(* CODESYS project Codesys_CtrlXCoreDriveConnectUtils
   Author: Riley Duffy
   Company: Open Source
   DefaultNamespace: DriveUtil
   Description: Library to Map Axis Information to it's name
   Title: Axis Info Mapping
   Version: 1.0.0

Project tree, tasks and I/O mapping:
  libraries: CXA_Datalayer, 2.6.20.0 (Bosch Rexroth AG); CXA_Flatbuffers, 0.1.3.2 (Bosch Rexroth AG); CXA_AutomationCore_fbs, 2.6.0.2717 (Bosch Rexroth AG); CXA_MotionCore_fbs, 2.6.0.1 (Bosch Rexroth AG); CXA_MotionSync_fbs, 2.6.0.4874 (Bosch Rexroth AG); CXA_CommonTypes, 1.18.1.0 (Bosch Rexroth AG); Standard, 3.5.18.0 (System); CXA_Utilities, 2.6.2.0 (Bosch Rexroth AG); ADT, 1.0.0 (Open Source); SysExcept, 3.5.17.0 (System)
  function block AxisInfoMap [ST]: Clear, GetAxisInfo, TryGetInfo, TryGetInfoFromAddr, TryPutInfo
  function block AxisInfoMap [ST]
  program AxisMapperPrg [ST]
  program AxisMapperPrg [ST]
  BoschSE_DriveInfoMapping.Sync
  commdata.all
  function block DriveParamBackup [ST]
  function block DriveParamRestore [ST]
  global variables GvlAxisInfo
  global variables GVLAxisInfoMap
  InternHelpers/
    AxisInfo/
      function block AxisInfoContainer [ST]: Get, GetPointer, GetSize, Put
      function block AxisInfoContainer [ST]
      data type typeAxisInfo
    function block AxisInfoMapper [ST]
    function block AxisInfoMapper [ST]
    function block BrowseAxis [ST]
    function block BrowseAxis [ST]
    function block comm_datalayer_DiagMoreInfo [ST]: _assign, _init, addKey, addValue, createDiagMoreInfo, endDiagMoreInfo, getKey, getKeyAsBytePtr, getRootAsDiagMoreInfo, getValue, getValueAsBytePtr, keysCompare, startDiagMoreInfo, verify, verifyDiagMoreInfo
    function block comm_datalayer_Diagnosis [ST]: _assign, _init, addCause, addDetailedDiagnosisCode, addDynamicDescription, addEntity, addMainDiagnosisCode, addMoreInfo, createCauseVector, createDiagnosis, createSortedmoreInfoVector, endDiagnosis, getCause, getCauseLength, getDetailedDiagnosisCode, getDynamicDescription, getDynamicDescriptionAsBytePtr, getEntity, getEntityAsBytePtr, getMainDiagnosisCode, getMoreInfo, getMoreInfoLength, getRootAsDiagnosis, startCauseVector, startDiagnosis, startMoreInfoVector, verify, verifyDiagnosis
    function block comm_datalayer_ProgramTask [ST]: _assign, _init, addId, addProgress, addProgressData, addProgressInfo, addResult, addState, createProgramTask, createSortedprogressDataVector, endProgramTask, getId, getIdAsBytePtr, getProgress, getProgressData, getProgressDataLength, getProgressInfo, getProgressInfoAsBytePtr, getResult, getRootAsProgramTask, getState, keysCompare, startProgramTask, startProgressDataVector, verify, verifyProgramTask
    data type comm_datalayer_ProgramTaskState
    function block comm_datalayer_ProgressData [ST]: _assign, _init, addKey, addValue, createProgressData, endProgressData, getKey, getKeyAsBytePtr, getRootAsProgressData, getValue, getValueAsBytePtr, keysCompare, startProgressData, verify, verifyProgressData
    function block comm_drive_ExportParFile_ExportParFile [ST]: _assign, _init, addBackupType, addFileName, createExportParFile, endExportParFile, getBackupType, getFileName, getFileNameAsBytePtr, getRootAsExportParFile, startExportParFile, verify, verifyExportParFile
    data type comm_drive_ExportParFile_ParametersType
    function block comm_drive_importParameter_ImportParameter [ST]: _assign, _init, addFileName, addSetIndex, createImportParameter, endImportParameter, getFileName, getFileNameAsBytePtr, getRootAsImportParameter, getSetIndex, startImportParameter, verify, verifyImportParameter
    Comparator/
      function block StringCompare [ST]: Compare
      function block StringCompare [ST]
      function block UdintCompare [ST]: Compare
      function block UdintCompare [ST]
    Containers/
      function block DeviceConnectNodeContainer [ST]: Get, GetPointer, GetSize, Put
      function block DeviceConnectNodeContainer [ST]
      function block HashDataContainer [ST]: Get, GetPointer, GetSize, Put
      function block HashDataContainer [ST]
      function block StringDataContainer [ST]: Get, GetPointer, GetSize, Put
      function block StringDataContainer [ST]
      function block UdintContainer [ST]: Get, GetPointer, GetSize, Put
      function block UdintContainer [ST]
    function block DCBrowseForFile [ST]
    data type EN_DRIVE_BACKUP_RESTORE_ERROR
    function block GetAllDriveConnectDevices [ST]
    function block GetAllDriveConnectDevices [ST]
    Hasher/
      function block UdintHash [ST]: Hash
      function block UdintHash [ST]
    function block InitAxisInfoMap [ST]
    function block InitAxisInfoMap [ST]
    function block MapDriveConnect [ST]
    function block MapDriveConnect [ST]
    function StrDecToUDINT [ST]
    function StringHexToUDINT [ST]
    function StringHexToUDINT [ST]
    data type typeDeviceConnectNode
    data type typeDeviceConnectNode
  libDriveUtil.Sync
  function block License_And_Use [ST]
  global variables Param
  global variables Param
  data type typeAxisInfo
*)

// typeAxisInfo
TYPE typeAxisInfo :
STRUCT
	sAxisName: STRING;
	sProfileName: STRING;
	udECatAddr: UDINT;
	sDriveConnectName: STRING;
	iDriveConnectSubDevice: UINT;
END_STRUCT
END_TYPE

// InternHelpers/comm_datalayer_ProgramTaskState
///automatically generated by the FlatBuffers compiler, do not modify
///comm\datalayer
{attribute 'qualified_only' := ''}
TYPE comm_datalayer_ProgramTaskState :
(
	/// task is pending and not been started
	pending := 0,
	/// task finished with failure
	failed := 1,
	/// task is successfully done
	done := 2,
	/// task is running
	running := 3
) BYTE;
END_TYPE

// InternHelpers/comm_drive_ExportParFile_ParametersType
///automatically generated by the FlatBuffers compiler, do not modify
///comm\drive\ExportParFile
{attribute 'qualified_only' := ''}
TYPE comm_drive_ExportParFile_ParametersType :
(
	All := 0,
	Backup := 1,
	Modified := 2
) UDINT;
END_TYPE

// InternHelpers/EN_DRIVE_BACKUP_RESTORE_ERROR
{attribute 'qualified_only' := ''}
{attribute 'strict' := ''}
TYPE EN_DRIVE_BACKUP_RESTORE_ERROR :
(
	OK := 0,
	RequestFailed := 1,
	ProgressReadFailed := 2,
	BackupFailed := 3,
	FileBrowseFailed := 4,
	FileExists := 5,
	DeleteFailed := 6,
	FileNotFound := 7,
	RestoreFailed := 8
);
END_TYPE

// InternHelpers/typeDeviceConnectNode
TYPE typeDeviceConnectNode :
STRUCT
	sNodeName: STRING;
	arSubDevices: ARRAY[0..4] OF STRING;
	uiNumbSubDevices: UINT;
END_STRUCT
END_TYPE

// InternHelpers/typeDeviceConnectNode
{attribute 'hide'}
TYPE typeDeviceConnectNode :
STRUCT
	sNodeName: STRING;
	arSubDevices: ARRAY[0..4] OF STRING;
	uiNumbSubDevices: UINT;
END_STRUCT
END_TYPE

// InternHelpers/AxisInfo/typeAxisInfo
TYPE typeAxisInfo :
STRUCT
	sAxisName: STRING;
	sProfileName: STRING;
	udECatAddr: UDINT;
	sDriveConnectName: STRING;
	iDriveConnectSubDevice: UINT;
END_STRUCT
END_TYPE

// GvlAxisInfo
{attribute 'qualified_only' := ''}
VAR_GLOBAL
	///Map with the Axis Name or EtherCat Address as Key. All Axis used in motion profile auto initialized
	Map: AxisInfoMap;
	///Axis found in the Motion App mapped
	bInitalized: BOOL;
	///Set true to run initialization again, useful if putting non Motion App Drives on map
	bReinitalize: BOOL;
	bClearMap: BOOL;
	///Error Occured during initialization
	Error: BOOL;
	///Only Valid if Error = TRUE
	ErrorID: ERROR_CODE;
	///Only Valid if Error = TRUE
	ErrorIdent: ERROR_STRUCT;
	///Only Valid if Error = TRUE
	ErrorStep: UINT;
END_VAR

// GVLAxisInfoMap
{attribute 'qualified_only'}
(* Interface to the library, Map contains the Drive Axis Info*)
VAR_GLOBAL
	Map : AxisInfoMap; 
	bInitalized :BOOL;
	bReinitalize : BOOL; 
	Error: BOOL;
	ErrorID: ERROR_CODE;
	ErrorIdent: ERROR_STRUCT;
	ErrorStep: UINT;
END_VAR

// Param
{attribute 'parameterlist' := ''}
{attribute 'qualified_only' := ''}
VAR_GLOBAL CONSTANT
	MAX_AXIS: UDINT := 10;
	USE_DRIVE_CONNECT: BOOL := TRUE;
END_VAR

// Param
{attribute 'qualified_only'}
VAR_GLOBAL CONSTANT
	MAX_AXIS : UDINT := 10; 
	USE_DRIVE_CONNECT : BOOL := TRUE; 
END_VAR

// AxisInfoMap
FUNCTION_BLOCK AxisInfoMap
VAR
	Values: AxisInfoContainer;
	Keys: StringDataContainer;
	StrHasher: StringHash;
	StrCompare: StringCompare;
	HashData: HashDataContainer;
	StrHashTable: HashTable := (KeyContainer := Keys, HashDataContainer := HashData, Compareator := StrCompare, Hasher := StrHasher);
	{attribute 'analysis' := '-33'}
	strMap: Map := (KeyContainer := StrHashTable, ValueContainer := Values);
	strValues: StringDataContainer;
	udintKeys: UdintContainer;
	udintHasher: UDintHash;
	udintCompare: UdintCompare;
	HashData2: HashDataContainer;
	UdintHashTable: HashTable := (KeyContainer := udintKeys, HashDataContainer := HashData2, Compareator := udintCompare, Hasher := udintHasher);
	{attribute 'analysis' := '-33'}
	UdintMap: Map := (KeyContainer := UdintHashTable, ValueContainer := strValues);
	stAxisInfo: typeAxisInfo;
END_VAR

METHOD INTERNAL Clear : BOOL
VAR_INPUT
END_VAR
strMap.Clear(); 
UdintMap.Clear();
END_METHOD

METHOD GetAxisInfo : REFERENCE TO typeAxisInfo
VAR_INPUT
	sAxisName: STRING;
END_VAR
strMap.Get(ADR(sAxisName), ADR(stAxisInfo)); 
GetAxisInfo REF= stAxisInfo;
END_METHOD

METHOD TryGetInfo : BOOL
VAR_INPUT
	sAxisName: STRING;
END_VAR
VAR_OUTPUT
	stAxisInfo: typeAxisInfo;
END_VAR
TryGetInfo := strMap.Get(adr(sAxisName),adr(stAxisInfo));
END_METHOD

METHOD TryGetInfoFromAddr : BOOL
VAR_INPUT
	Addr: UDINT;
END_VAR
VAR_OUTPUT
	stAxisInfo: typeAxisInfo;
END_VAR
VAR
	_sAxisName: STRING;
END_VAR
IF UdintMap.Get(ADR(addr),ADR(_sAxisName)) THEN 
	TryGetInfoFromAddr := StrMap.Get(ADR(_sAxisName),ADR(stAxisInfo)); 
ELSE 
	TryGetInfoFromAddr := FALSE; 
END_IF
END_METHOD

METHOD TryPutInfo : BOOL
VAR_INPUT
	sAxisName: STRING;
	stAxisInfo: typeAxisInfo;
END_VAR
TryPutInfo := strMap.Put(ADR(sAxisName),ADR(stAxisInfo)); 
IF stAxisInfo.udECatAddr <> 0 THEN 
	UdintMap.Put(ADR(stAxisInfo.udECatAddr),ADR(sAxisName)); 
END_IF
END_METHOD

END_FUNCTION_BLOCK

// AxisInfoMap
///Axis Info Map used to relate Ethercat Addresses and DeviceConnect Names to axis Name
FUNCTION_BLOCK AxisInfoMap
VAR
	Values: AxisInfoContainer;
	Keys: StringDataContainer;
	StrHasher: StringHash;
	StrCompare: StringCompare;
	HashData: HashDataContainer;
	StrHashTable: HashTable := (KeyContainer := Keys, HashDataContainer := HashData, Compareator := StrCompare, Hasher := StrHasher);
	{attribute 'analysis' := '-33'}
	strMap: Map := (KeyContainer := StrHashTable, ValueContainer := Values);
	strValues: StringDataContainer;
	udintKeys: UdintContainer;
	udintHasher: UDintHash;
	udintCompare: UdintCompare;
	HashData2: HashDataContainer;
	UdintHashTable: HashTable := (KeyContainer := udintKeys, HashDataContainer := HashData2, Compareator := udintCompare, Hasher := udintHasher);
	{attribute 'analysis' := '-33'}
	UdintMap: Map := (KeyContainer := UdintHashTable, ValueContainer := strValues);
	stAxisInfo: typeAxisInfo;
END_VAR

END_FUNCTION_BLOCK

// InternHelpers/AxisInfo/AxisInfoContainer
{attribute 'hide'}
FUNCTION_BLOCK AxisInfoContainer IMPLEMENTS iDataContainer
VAR CONSTANT
	_size : UDINT := TO_UDINT(TO_REAL(Param.MAX_AXIS)* 1.3);
END_VAR 
VAR
	_arBacking: ARRAY[0.._size -1] OF typeAxisInfo;
	_pData: POINTER TO typeAxisInfo;
END_VAR

{attribute 'hide'}
METHOD Get : BOOL
VAR_INPUT
	index: UDINT;
	pData: PVoid;
END_VAR
_pData := pData; 
IF index < _size THEN 
	_pData^ := _arBacking[index]; 
	Get := TRUE;
ELSE 
	Get := FALSE; 
END_IF
END_METHOD

{attribute 'hide'}
METHOD GetPointer : PVoid
VAR_INPUT
	index: UDINT;
END_VAR
IF index < _size THEN 
	GetPointer:= ADR(_arBacking[index]); 
ELSE 
	GetPointer := 0; 
END_IF
END_METHOD

{attribute 'hide'}
METHOD GetSize : UDINT
GetSize := _size;
END_METHOD

{attribute 'hide'}
METHOD Put : BOOL
VAR_INPUT
	index: UDINT;
	pData: PVoid;
END_VAR
_pData := pData; 
IF index < _size THEN 
	_arBacking[index] := _pData^; 
	Put := TRUE; 
ELSE 
	Put := FALSE; 
END_IF
END_METHOD

END_FUNCTION_BLOCK

// InternHelpers/AxisInfo/AxisInfoContainer
FUNCTION_BLOCK AxisInfoContainer IMPLEMENTS iDataContainer
VAR CONSTANT
	_size: UDINT := ANY_TO_UDINT((ANY_TO_REAL(Param.MAX_AXIS) * 1.3));
END_VAR
VAR
	_arBacking: ARRAY[0..(_size - 1)] OF typeAxisInfo;
	_pData: POINTER TO typeAxisInfo;
END_VAR

END_FUNCTION_BLOCK

// InternHelpers/Containers/StringDataContainer
{attribute 'hide'}
{attribute 'no_check' := ''}
FUNCTION_BLOCK StringDataContainer IMPLEMENTS iDataContainer
VAR CONSTANT
	_size : UDINT := TO_UDINT(TO_REAL(Param.MAX_AXIS)* 1.3);
END_VAR 
VAR
	_arBacking: ARRAY[0.._size -1] OF STRING(255);
	_pData: POINTER TO String(255);
END_VAR

{attribute 'hide'}
{attribute 'no_check' := ''}
METHOD Get : BOOL
VAR_INPUT
	index: UDINT;
	pData: PVoid;
END_VAR
_pData := pData; 
IF index < _size THEN 
	_pData^ := _arBacking[index]; 
	Get := TRUE;
ELSE 
	Get := FALSE; 
END_IF
END_METHOD

{attribute 'hide'}
{attribute 'no_check' := ''}
METHOD GetPointer : PVoid
VAR_INPUT
	index: UDINT;
END_VAR
IF index < _size THEN 
	GetPointer:= ADR(_arBacking[index]); 
ELSE 
	GetPointer := 0; 
END_IF
END_METHOD

{attribute 'hide'}
METHOD GetSize : UDINT
GetSize := _size;
END_METHOD

{attribute 'hide'}
{attribute 'no_check' := ''}
METHOD Put : BOOL
VAR_INPUT
	index: UDINT;
	pData: PVoid;
END_VAR
_pData := pData; 
IF index < _size THEN 
	_arBacking[index] := _pData^; 
	Put := TRUE; 
ELSE 
	Put := FALSE; 
END_IF
END_METHOD

END_FUNCTION_BLOCK

// InternHelpers/Containers/StringDataContainer
{attribute 'no_check' := ''}
FUNCTION_BLOCK StringDataContainer IMPLEMENTS iDataContainer
VAR CONSTANT
	_size: UDINT := ANY_TO_UDINT((ANY_TO_REAL(Param.MAX_AXIS) * 1.3));
END_VAR
VAR
	_arBacking: ARRAY[0..(_size - 1)] OF STRING(255);
	_pData: POINTER TO STRING(255);
END_VAR

END_FUNCTION_BLOCK

// InternHelpers/Comparator/StringCompare
{attribute 'hide'}
{attribute 'no_check' := ''}
FUNCTION_BLOCK StringCompare IMPLEMENTS iCompare

{attribute 'hide'}
METHOD Compare : INT
VAR_INPUT
	pData1: PVoid;
	pData2: PVoid;
END_VAR
VAR
	pStr1: POINTER TO STRING := pData1;
	pStr2: POINTER TO STRING := pData2;
END_VAR
IF pStr1^ = pStr2^ THEN 
	Compare := 0; 
ELSE 
	Compare := 1; 
END_IF
END_METHOD

END_FUNCTION_BLOCK

// InternHelpers/Comparator/StringCompare
{attribute 'no_check' := ''}
FUNCTION_BLOCK StringCompare IMPLEMENTS iCompare

END_FUNCTION_BLOCK

// InternHelpers/Containers/HashDataContainer
{attribute 'no_check' := ''}
FUNCTION_BLOCK HashDataContainer IMPLEMENTS iDataContainer
VAR CONSTANT
	_size: UDINT := ANY_TO_UDINT((ANY_TO_REAL(Param.MAX_AXIS) * 1.3));
END_VAR
VAR
	_arBacking: ARRAY[0..(_size - 1)] OF HashData;
	_pData: POINTER TO HashData;
END_VAR

{attribute 'no_check' := ''}
METHOD Get : BOOL
VAR_INPUT
	index: UDINT;
	pData: PVoid;
END_VAR
_pData := pData; 
IF index < _size THEN 
	_pData^ := _arBacking[index]; 
	Get := TRUE;
ELSE 
	Get := FALSE; 
END_IF
END_METHOD

{attribute 'no_check' := ''}
METHOD GetPointer : PVoid
VAR_INPUT
	index: UDINT;
END_VAR
IF index < _size THEN 
	GetPointer:= ADR(_arBacking[index]); 
ELSE 
	GetPointer := 0; 
END_IF
END_METHOD

METHOD GetSize : UDINT
GetSize := _size;
END_METHOD

{attribute 'no_check' := ''}
METHOD Put : BOOL
VAR_INPUT
	index: UDINT;
	pData: PVoid;
END_VAR
_pData := pData; 
IF index < _size THEN 
	_arBacking[index] := _pData^; 
	Put := TRUE; 
ELSE 
	Put := FALSE; 
END_IF
END_METHOD

END_FUNCTION_BLOCK

// InternHelpers/Containers/HashDataContainer
{attribute 'hide'}
{attribute 'no_check' := ''}
FUNCTION_BLOCK HashDataContainer IMPLEMENTS iDataContainer
VAR CONSTANT
	_size : UDINT := TO_UDINT(TO_REAL(Param.MAX_AXIS)* 1.3);
END_VAR 
VAR
	_arBacking: ARRAY[0.._size -1] OF HashData;
	_pData: POINTER TO HashData;
END_VAR

END_FUNCTION_BLOCK

// InternHelpers/Containers/UdintContainer
{attribute 'hide'}
{attribute 'no_check' := ''}
FUNCTION_BLOCK UdintContainer IMPLEMENTS iDataContainer
VAR CONSTANT
	_size : UDINT := TO_UDINT(TO_REAL(Param.MAX_AXIS)* 1.3);
END_VAR 
VAR
	_arBacking: ARRAY[0.._size -1] OF UDINT;
	_pData: POINTER TO UDINT;
END_VAR

{attribute 'hide'}
{attribute 'no_check' := ''}
METHOD Get : BOOL
VAR_INPUT
	index: UDINT;
	pData: PVoid;
END_VAR
_pData := pData; 
IF index < _size THEN 
	_pData^ := _arBacking[index]; 
	Get := TRUE;
ELSE 
	Get := FALSE; 
END_IF
END_METHOD

{attribute 'hide'}
{attribute 'no_check' := ''}
METHOD GetPointer : PVoid
VAR_INPUT
	index: UDINT;
END_VAR
IF index < _size THEN 
	GetPointer:= ADR(_arBacking[index]); 
ELSE 
	GetPointer := 0; 
END_IF
END_METHOD

{attribute 'hide'}
METHOD GetSize : UDINT
GetSize := _size;
END_METHOD

{attribute 'hide'}
{attribute 'no_check' := ''}
METHOD Put : BOOL
VAR_INPUT
	index: UDINT;
	pData: PVoid;
END_VAR
_pData := pData; 
IF index < _size THEN 
	_arBacking[index] := _pData^; 
	Put := TRUE; 
ELSE 
	Put := FALSE; 
END_IF
END_METHOD

END_FUNCTION_BLOCK

// InternHelpers/Containers/UdintContainer
{attribute 'no_check' := ''}
FUNCTION_BLOCK UdintContainer IMPLEMENTS iDataContainer
VAR CONSTANT
	_size: UDINT := ANY_TO_UDINT((ANY_TO_REAL(Param.MAX_AXIS) * 1.3));
END_VAR
VAR
	_arBacking: ARRAY[0..(_size - 1)] OF UDINT;
	_pData: POINTER TO UDINT;
END_VAR

END_FUNCTION_BLOCK

// InternHelpers/Hasher/UdintHash
{attribute 'hide'}
{attribute 'no_check' := ''}
FUNCTION_BLOCK UdintHash IMPLEMENTS iHash

{attribute 'hide'}
METHOD Hash : LINT
VAR_INPUT
	pData: pVoid;
END_VAR
VAR
	ptrUdint: POINTER TO UDINT := pData;
END_VAR
Hash := TO_LINT(ptrUdint^);
END_METHOD

END_FUNCTION_BLOCK

// InternHelpers/Hasher/UdintHash
{attribute 'no_check' := ''}
FUNCTION_BLOCK UdintHash IMPLEMENTS iHash

END_FUNCTION_BLOCK

// InternHelpers/Comparator/UdintCompare
{attribute 'hide'}
{attribute 'no_check' := ''}
FUNCTION_BLOCK UdintCompare IMPLEMENTS iCompare

{attribute 'hide'}
METHOD Compare : INT
VAR_INPUT
	pData1: PVoid;
	pData2: PVoid;
END_VAR
VAR
	pUdint1: POINTER TO UDINT := pData1;
	pUdint2: POINTER TO UDINT := pData2;
END_VAR
IF pUdint1^ = pUdint2^ THEN 
	Compare := 0; 
ELSIF pUdint1^ > pUdint2^ THEN 
	Compare := 1; 
ELSE
	Compare := -1; 
END_IF
END_METHOD

END_FUNCTION_BLOCK

// InternHelpers/Comparator/UdintCompare
{attribute 'no_check' := ''}
FUNCTION_BLOCK UdintCompare IMPLEMENTS iCompare

END_FUNCTION_BLOCK

// AxisMapperPrg
PROGRAM AxisMapperPrg
VAR
	_instAxisMapper: AxisInfoMapper;
	_dlBrowse: CXA_DATALAYER.DL_BrowseNode;
	_sBrowseDevices: STRING(255) := 'devices/drives';
	_bReady: BOOL;
	_fbBootDelay : TON; 
	_bFirstScan : BOOL := TRUE; 
END_VAR

_fbBootDelay(IN := NOT _bFirstScan, PT := T#10s); 
_bFirstScan := FALSE; 
IF NOT _fbBootDelay.Q THEN 
	RETURN
END_IF
IF PARAM.USE_DRIVE_CONNECT AND NOT _bReady THEN 
	_dlBrowse(execute := NOT _bReady, 
			  NodeName := _sBrowseDevices); 
	IF _dlBrowse.Done AND _dlBrowse.ChildPtr = 0 THEN 
		_dlBrowse(execute := FALSE);
	ELSIF _dlBrowse.Done THEN 
		_bReady := TRUE; 
	END_IF
END_IF
IF NOT _bReady THEN 
	RETURN; 
END_IF
_instAxisMapper(bExecute := GvlAxisInfo.bReinitalize OR (NOT GvlAxisInfo.bInitalized AND NOT GvlAxisInfo.Error),
				bUseDriveConnect := Param.USE_DRIVE_CONNECT, 
				instAxisInfoMap := GvlAxisInfo.Map); 
IF _instAxisMapper.bDone THEN 
	GvlAxisInfo.bInitalized := TRUE; 
END_IF
IF GvlAxisInfo.bReinitalize THEN 
	GvlAxisInfo.Error := FALSE; 
END_IF
IF _instAxisMapper.bActive THEN 
	GvlAxisInfo.bInitalized := FALSE; 
END_IF
IF GVLAxisInfo.bClearMap THEN 
	GVLAxisInfo.Map.Clear();
	GvlAxisInfo.bInitalized := FALSE; 
END_IF
IF _instAxisMapper.bError THEN 
	GvlAxisInfo.Error := TRUE; 
END_IF 
IF _instAxisMapper.bError THEN 
	GvlAxisInfo.ErrorID := _instAxisMapper.ErrorID; 
	GvlAxisInfo.ErrorIdent := _instAxisMapper.ErrorIdent; 
	GvlAxisInfo.ErrorStep := _instAxisMapper.ErrorStep; 
END_IF

END_PROGRAM

// AxisMapperPrg
(* Program that searches the configured axis in CtrxCore and gets 
   their Ethercat addresses and Drive Connect info (serial number, drive index)*)
PROGRAM AxisMapperPrg
VAR
	_instAxisMapper : AxisInfoMapper; 
END_VAR
VAR_OUTPUT
	
END_VAR

_instAxisMapper(bExecute := GvlAxisInfoMap.bReinitalize OR NOT GvlAxisInfoMap.bInitalized,
				bUseDriveConnect := Param.USE_DRIVE_CONNECT, 
				instAxisInfoMap := GvlAxisInfoMap.Map); 
IF _instAxisMapper.bDone THEN 
	GvlAxisInfoMap.bInitalized := TRUE; 
END_IF
IF _instAxisMapper.bActive THEN 
	GvlAxisInfoMap.bInitalized := FALSE; 
END_IF

GVLAxisInfoMap.Error := _instAxisMapper.bError; 
IF _instAxisMapper.bError THEN 
	GVLAxisInfoMap.ErrorID := _instAxisMapper.ErrorID; 
	GVLAxisInfoMap.ErrorIdent := _instAxisMapper.ErrorIdent; 
	GVLAxisInfoMap.ErrorStep := _instAxisMapper.ErrorStep; 
END_IF

END_PROGRAM

// InternHelpers/AxisInfoMapper
FUNCTION_BLOCK AxisInfoMapper
VAR_INPUT
	bExecute: BOOL;
	bUseDriveConnect: BOOL;
END_VAR
VAR_IN_OUT
	instAxisInfoMap: AxisInfoMap;
END_VAR
VAR_OUTPUT
	bDone: BOOL;
	bActive: BOOL;
	bError: BOOL;
	ErrorID: ERROR_CODE;
	ErrorIdent: ERROR_STRUCT;
	ErrorStep: UINT;
END_VAR
VAR
	_uiNextState: UINT;
	_uiState: UINT;
	_instInitAxisInfo: InitAxisInfoMap;
	_instMapDriveConnect: MapDriveConnect;
END_VAR
VAR CONSTANT
	IDLE: UINT := 0;
	INIT_AXIS_INFO_MAP: UINT := 1;
	MAP_DRIVE_CONNECT: UINT := 2;
	DONE: UINT := 3;
	ERROR: UINT := 4;
END_VAR

_uiNextState := _uiState; 
CASE _uiState OF 
	IDLE : 
		IF bExecute THEN 
			_uiNextState := INIT_AXIS_INFO_MAP;  
		END_IF
	INIT_AXIS_INFO_MAP: 
		IF _instInitAxisInfo.bError THEN 
			bError := TRUE; 
			ERRORID := _instInitAxisInfo.enErrorID; 
			ErrorIdent := _instInitAxisInfo.enErrorIdent; 
			ErrorStep := INIT_AXIS_INFO_MAP; 
			_uiNextState := ERROR; 
		ELSIF _instInitAxisInfo.bDone THEN 
			IF bUseDriveConnect THEN 
				_uiNextState := MAP_DRIVE_CONNECT; 
			ELSE 
				_uiNextState := DONE; 
			END_IF
		END_IF
	MAP_DRIVE_CONNECT: 
		IF _instMapDriveConnect.bError THEN 
			bError := TRUE; 
			ERRORID := _instMapDriveConnect.enErrorID; 
			ErrorIdent := _instMapDriveConnect.stErrorIdent; 
			ErrorStep := INIT_AXIS_INFO_MAP; 
			_uiNextState := ERROR; 
		ELSIF _instMapDriveConnect.bDone THEN 
			_uiNextState := DONE; 
		END_IF
	DONE,ERROR : 
		IF NOT bExecute THEN 
			_uiNextState := IDLE; 
		END_IF
END_CASE
_uiState := _uiNextState; 
_instInitAxisInfo(bExecute := _uiState = INIT_AXIS_INFO_MAP, 
				  instAxisInfoMap := instAxisInfoMap); 
_instMapDriveConnect(bExecute := _uiState = MAP_DRIVE_CONNECT, 
					 instAxisInfoMap := instAxisInfoMap); 
bDone := _uiState = DONE; 
bError := _uiState = ERROR; 
bActive := _uiState <> IDLE AND _uiState <> DONE AND _uiState <> ERROR;

END_FUNCTION_BLOCK

// InternHelpers/AxisInfoMapper
{attribute 'hide'}
(*Handles the sate logic for drive info search*)
FUNCTION_BLOCK AxisInfoMapper
VAR_INPUT
	bExecute : BOOL; 
	bUseDriveConnect : BOOL; 
END_VAR
VAR_IN_OUT 
	instAxisInfoMap : AxisInfoMap; 
END_VAR
VAR_OUTPUT
	bDone     : BOOL; 
	bActive   : BOOL; 
	bError    : BOOL;  
	ErrorID: ERROR_CODE;
	ErrorIdent: ERROR_STRUCT;
	ErrorStep: UINT;
END_VAR
VAR
	_uiNextState : UINT;
	_uiState     : UINT; 
	_instInitAxisInfo : InitAxisInfoMap; 
	_instMapDriveConnect : MapDriveConnect;  
END_VAR
VAR CONSTANT
	IDLE : UINT := 0; 
	INIT_AXIS_INFO_MAP : UINT := 1; 
	MAP_DRIVE_CONNECT : UINT := 2; 
	DONE              : UINT := 3; 
	ERROR			  : UINT := 4; 
END_VAR

_uiNextState := _uiState; 
CASE _uiState OF 
	IDLE : 
		IF bExecute THEN 
			_uiNextState := INIT_AXIS_INFO_MAP; 
			instAxisInfoMap.Clear(); 
		END_IF
	INIT_AXIS_INFO_MAP: 
		IF _instInitAxisInfo.bError THEN 
			bError := TRUE; 
			ERRORID := _instInitAxisInfo.enErrorID; 
			ErrorIdent := _instInitAxisInfo.enErrorIdent; 
			ErrorStep := INIT_AXIS_INFO_MAP; 
			_uiNextState := ERROR; 
		ELSIF _instInitAxisInfo.bDone THEN 
			IF bUseDriveConnect THEN 
				_uiNextState := MAP_DRIVE_CONNECT; 
			ELSE 
				_uiNextState := DONE; 
			END_IF
		END_IF
	MAP_DRIVE_CONNECT: 
		IF _instMapDriveConnect.bError THEN 
			bError := TRUE; 
			ERRORID := _instMapDriveConnect.enErrorID; 
			ErrorIdent := _instMapDriveConnect.stErrorIdent; 
			ErrorStep := INIT_AXIS_INFO_MAP; 
			_uiNextState := MAP_DRIVE_CONNECT; 
		ELSIF _instInitAxisInfo.bDone THEN 
			_uiNextState := DONE; 
		END_IF
	DONE,ERROR : 
		IF NOT bExecute THEN 
			_uiNextState := IDLE; 
		END_IF
END_CASE
_uiState := _uiNextState; 
_instInitAxisInfo(bExecute := _uiState = INIT_AXIS_INFO_MAP, 
				  instAxisInfoMap := instAxisInfoMap); 
_instMapDriveConnect(bExecute := _uiState = MAP_DRIVE_CONNECT, 
					 instAxisInfoMap := instAxisInfoMap); 
bDone := _uiState = DONE; 
bError := _uiState = ERROR; 
bActive := _uiState <> IDLE AND _uiState <> DONE AND _uiState <> ERROR;

END_FUNCTION_BLOCK

// InternHelpers/InitAxisInfoMap
FUNCTION_BLOCK InitAxisInfoMap
VAR_INPUT
	bExecute: BOOL;
END_VAR
VAR_OUTPUT
	bDone: BOOL;
	bError: BOOL;
	bActive: BOOL;
	enErrorID: ERROR_CODE;
	enErrorIdent: ERROR_STRUCT;
	uiErrorStep: UINT;
END_VAR
VAR_IN_OUT
	instAxisInfoMap: AxisInfoMap;
END_VAR
VAR
	_instBrowseAxis: BrowseAxis;
	_instDLReadAxis: DL_ReadNodeValue;
	_instDLReadProfile: DL_ReadNodeValue;
	_instDLNodeAxis: DL_NodeValue;
	_instDLNodeProfile: DL_NodeValue;
	_axConfig: motion_core_fbtypes_AxsCfg;
	_axProfile: comm_axisprofile_fbtypes_profileConfig;
	_stAxisInfo: typeAxisInfo;
	_stDefualtAxisInfo: typeAxisInfo;
	_uiNextState: UINT;
	_uiState: UINT;
	_axisIndex: UDINT;
	_arAxisNames: ARRAY[0..Param.MAX_AXIS] OF STRING;
	_sAxisNode: STRING(255);
	_sProfileNode: STRING(255);
END_VAR
VAR CONSTANT
	IDLE: UINT := 0;
	BROWSE_AXIS: UINT := 1;
	READ_DL_AXIS_CFG: UINT := 2;
	READ_DL_PROFILE: UINT := 3;
	UPDATE_MAP: UINT := 4;
	DONE: UINT := 5;
	ERROR: UINT := 6;
END_VAR

_uiNextState := _uiState; 
CASE _uiState OF 
	IDLE: 
		IF bExecute THEN 
			_uiNextState := BROWSE_AXIS; 
		END_IF
	BROWSE_AXIS: 
		IF _instBrowseAxis.Error THEN 
			_uiNextState := ERROR; 
			enErrorID := _instBrowseAxis.ErrorID; 
			enErrorIdent := _instBrowseAxis.ErrorIdent; 
			uiErrorStep := BROWSE_AXIS; 
		ELSIF _instBrowseAxis.Done THEN 
			_uiNextState := READ_DL_AXIS_CFG; 
		END_IF
	READ_DL_AXIS_CFG: 
		IF _instDLReadAxis.Error THEN 
			_uiNextState := ERROR; 
			enErrorID := _instDLReadAxis.ErrorID; 
			enErrorIdent := _instDLReadAxis.ErrorIdent; 
			uiErrorStep := READ_DL_AXIS_CFG; 
		ELSIF _instDLReadAxis.Done THEN 
			_axConfig.getRootAsAxsCfg(_instDLNodeAxis.GetData(),_instDLNodeAxis.GetSize()); 
			IF _axConfig.getAxisProfileName() <> '' THEN 
				_uiNextState := READ_DL_PROFILE;
			ELSE 
				_uiNextState := UPDATE_MAP; 
			END_IF  
		END_IF
	READ_DL_PROFILE: 
		IF _instDLReadProfile.Error THEN 
			_uiNextState := ERROR; 
		ELSIF _instDLReadProfile.Done THEN 
			_uiNextState := UPDATE_MAP; 
			enErrorID := _instDLReadProfile.ErrorID; 
			enErrorIdent := _instDLReadProfile.ErrorIdent; 
			uiErrorStep := READ_DL_PROFILE; 
		END_IF
	UPDATE_MAP: 
		_axisIndex := _axisIndex + 1; 
		IF _axisIndex < _instBrowseAxis.NbAxis THEN 
			_uiNextState := READ_DL_AXIS_CFG; 
		ELSE 
			_uiNextState := DONE; 
		END_IF
	DONE,ERROR: 
		IF NOT bExecute THEN 
			_uiNextState := IDLE; 
		END_IF
END_CASE
_uiState := _uiNextState; 
CASE _uiState OF 
	IDLE: 
		_axisIndex := 0; 
	BROWSE_AXIS: 
		;
	READ_DL_AXIS_CFG: 
		_stAxisInfo := _stDefualtAxisInfo;
		_sAxisNode := Concat('motion/axs/',_arAxisNames[_axisIndex]); 
		_sAxisNode := Concat(_sAxisNode,'/cfg');  
	READ_DL_PROFILE:
		_sProfileNode := Concat('axisprofile/profiles/', _axConfig.getAxisProfileName()); 
		_sProfileNode := Concat(_sProfileNode,'/cfg'); 
	UPDATE_MAP: 
		_axProfile.getRootAsprofileConfig(_instDLNodeProfile.getData(), _instDLNodeProfile.GetSize());
		_stAxisInfo.sAxisName := _arAxisNames[_axisIndex]; 
		_stAxisInfo.sProfileName :=  _axConfig.getAxisProfileName(); 
		IF _stAxisInfo.sProfileName <> '' THEN 
			_stAxisInfo.udECatAddr := _axProfile.getDeviceAddress(); 
		END_IF; 
		instAxisInfoMap.TryPutInfo(_arAxisNames[_axisIndex],_stAxisInfo, TRUE); 
	DONE,ERROR: 
		IF NOT bExecute THEN 
			_uiNextState := IDLE; 
		END_IF
END_CASE
_instBrowseAxis(Execute := _uiState = BROWSE_AXIS, 
				Axis := _arAxisNames); 
_instDLReadAxis(Execute := _uiState = READ_DL_AXIS_CFG, 
				NodeName := _sAxisNode,
				NodeValue := _instDLNodeAxis); 
_instDLReadProfile(Execute := _uiState = READ_DL_PROFILE, 
				   NodeName := _sProfileNode, 
				   NodeValue := _instDLNodeProfile); 
bDone := _uiState = DONE; 
bError := _uiState = ERROR; 
bActive := _uiState <> DONE AND _uiState <> IDLE AND _uiState <> ERROR;

END_FUNCTION_BLOCK

// InternHelpers/InitAxisInfoMap
{attribute 'hide'}
(* Buids the map for Axis Info by browsing for axis -> getting Ethercat info from profile
   Browse Drive Connect, match Ethercat addreess to Ethercat address parameter*) 
FUNCTION_BLOCK InitAxisInfoMap
VAR_INPUT
	bExecute: BOOL;
END_VAR
VAR_OUTPUT
	bDone: BOOL;
	bError: BOOL;
	bActive: BOOL;
	enErrorID: ERROR_CODE;
	enErrorIdent: ERROR_STRUCT;
	uiErrorStep: UINT;
END_VAR
VAR_IN_OUT
	instAxisInfoMap: AxisInfoMap;
END_VAR
VAR
	_instBrowseAxis: BrowseAxis;
	_instDLReadAxis: DL_ReadNodeValue;
	_instDLReadProfile: DL_ReadNodeValue;
	_instDLNodeAxis: DL_NodeValue;
	_instDLNodeProfile: DL_NodeValue;
	_axConfig: motion_core_fbtypes_AxsCfg;
	_axProfile: comm_axisprofile_fbtypes_profileConfig;
	_stAxisInfo: typeAxisInfo;
	_stDefualtAxisInfo: typeAxisInfo;
	_uiNextState: UINT;
	_uiState: UINT;
	_axisIndex: UDINT;
	_arAxisNames: ARRAY[0..Param.MAX_AXIS] OF STRING;
	_sAxisNode: STRING(255);
	_sProfileNode: STRING(255);
END_VAR
VAR CONSTANT
	IDLE: UINT := 0;
	BROWSE_AXIS: UINT := 1;
	READ_DL_AXIS_CFG: UINT := 2;
	READ_DL_PROFILE: UINT := 3;
	UPDATE_MAP: UINT := 4;
	DONE: UINT := 5;
	ERROR: UINT := 6;
END_VAR

_uiNextState := _uiState; 
CASE _uiState OF 
	IDLE: 
		IF bExecute THEN 
			_uiNextState := BROWSE_AXIS; 
		END_IF
	BROWSE_AXIS: 
		IF _instBrowseAxis.Error THEN 
			_uiNextState := ERROR; 
			enErrorID := _instBrowseAxis.ErrorID; 
			enErrorIdent := _instBrowseAxis.ErrorIdent; 
			uiErrorStep := BROWSE_AXIS; 
		ELSIF _instBrowseAxis.Done THEN 
			_uiNextState := READ_DL_AXIS_CFG; 
		END_IF
	READ_DL_AXIS_CFG: 
		IF _instDLReadAxis.Error THEN 
			_uiNextState := ERROR; 
			enErrorID := _instDLReadAxis.ErrorID; 
			enErrorIdent := _instDLReadAxis.ErrorIdent; 
			uiErrorStep := READ_DL_AXIS_CFG; 
		ELSIF _instDLReadAxis.Done THEN 
			_axConfig.getRootAsAxsCfg(_instDLNodeAxis.GetData(),_instDLNodeAxis.GetSize()); 
			IF _axConfig.getAxisProfileName() <> '' THEN 
				_uiNextState := READ_DL_PROFILE;
			ELSE 
				_uiNextState := UPDATE_MAP; 
			END_IF  
		END_IF
	READ_DL_PROFILE: 
		IF _instDLReadProfile.Error THEN 
			_uiNextState := ERROR; 
		ELSIF _instDLReadProfile.Done THEN 
			_uiNextState := UPDATE_MAP; 
			enErrorID := _instDLReadProfile.ErrorID; 
			enErrorIdent := _instDLReadProfile.ErrorIdent; 
			uiErrorStep := READ_DL_PROFILE; 
		END_IF
	UPDATE_MAP: 
		_axisIndex := _axisIndex + 1; 
		IF _axisIndex < _instBrowseAxis.NbAxis THEN 
			_uiNextState := READ_DL_AXIS_CFG; 
		ELSE 
			_uiNextState := DONE; 
		END_IF
	DONE,ERROR: 
		IF NOT bExecute THEN 
			_uiNextState := IDLE; 
		END_IF
END_CASE
_uiState := _uiNextState; 
CASE _uiState OF 
	IDLE: 
		_axisIndex := 0; 
	BROWSE_AXIS: 
		;
	READ_DL_AXIS_CFG: 
		_stAxisInfo := _stDefualtAxisInfo;
		_sAxisNode := Concat('motion/axs/',_arAxisNames[_axisIndex]); 
		_sAxisNode := Concat(_sAxisNode,'/cfg');  
	READ_DL_PROFILE:
		_sProfileNode := Concat('axisprofile/profiles/', _axConfig.getAxisProfileName()); 
		_sProfileNode := Concat(_sProfileNode,'/cfg'); 
	UPDATE_MAP: 
		_axProfile.getRootAsprofileConfig(_instDLNodeProfile.getData(), _instDLNodeProfile.GetSize());
		_stAxisInfo.sAxisName := _arAxisNames[_axisIndex]; 
		_stAxisInfo.sProfileName :=  _axConfig.getAxisProfileName(); 
		IF _stAxisInfo.sProfileName <> '' THEN 
			_stAxisInfo.udECatAddr := _axProfile.getDeviceAddress(); 
		END_IF; 
		instAxisInfoMap.TryPutInfo(_arAxisNames[_axisIndex],_stAxisInfo); 
	DONE,ERROR: 
		IF NOT bExecute THEN 
			_uiNextState := IDLE; 
		END_IF
END_CASE
_instBrowseAxis(Execute := _uiState = BROWSE_AXIS, 
				Axis := _arAxisNames); 
_instDLReadAxis(Execute := _uiState = READ_DL_AXIS_CFG, 
				NodeName := _sAxisNode,
				NodeValue := _instDLNodeAxis); 
_instDLReadProfile(Execute := _uiState = READ_DL_PROFILE, 
				   NodeName := _sProfileNode, 
				   NodeValue := _instDLNodeProfile); 
bDone := _uiState = DONE; 
bError := _uiState = ERROR; 
bActive := _uiState <> DONE AND _uiState <> IDLE AND _uiState <> ERROR;

END_FUNCTION_BLOCK

// InternHelpers/BrowseAxis
{attribute 'hide'}
{attribute 'no_assign' := ''}
(*Looks at all Axis configured in CtrxCore*)
FUNCTION_BLOCK BrowseAxis
VAR_INPUT
	Execute: BOOL;
END_VAR
VAR_OUTPUT
	Done: BOOL;
	Active: BOOL;
	Error: BOOL;
	ErrorID: ERROR_CODE;
	ErrorIdent: ERROR_STRUCT;
	NbAxis: UDINT;
END_VAR
VAR_IN_OUT
	Axis: ARRAY[*] OF STRING;
END_VAR
VAR
	_browseNode : DL_BROWSENODE; 
	_diArrayIndex : DINT; 
END_VAR

// example to browse all existing axisprofile 

// call fb, to browse for all configured axisprofile
_browseNode(
	Execute:= Execute, 
	Active=> Active, 
	Error=> Error, 
	ErrorID=> ErrorID, 
	ErrorIdent=> ErrorIdent, 
	NodeName:= 'motion/axs');
	
// check for done
IF _browseNode.Done THEN
	// check, if array size is large enough for the returned 
	IF (UDINT_TO_DINT(_browseNode.ChildNum) > (UPPER_BOUND(Axis, 1)-LOWER_BOUND(Axis, 1))) THEN 
		// array size not large enough => error
		Error:= TRUE;
		ErrorIdent.Table:= USER1_TABLE;
 		ErrorIdent.Additional1:= 16#0E0F0001; 
		ErrorIdent.Additional2:= 16#00000000;  
	ELSE 	
		// array size large enough => assign values
	  	FOR _diArrayIndex:= 0 TO (UPPER_BOUND(Axis, 1)-LOWER_BOUND(Axis, 1)) DO
			Axis[LOWER_BOUND(Axis, 1)+_diArrayIndex]:= _browseNode.GetChildName(Index:= DINT_TO_UDINT(_diArrayIndex));
		END_FOR
		// number of axis
		NbAxis:= _browseNode.ChildNum;
	END_IF
END_IF
// actualise output done
Done:= _browseNode.Done AND NOT Error;

END_FUNCTION_BLOCK

// InternHelpers/BrowseAxis
{attribute 'no_assign' := ''}
FUNCTION_BLOCK BrowseAxis
VAR_INPUT
	Execute: BOOL;
END_VAR
VAR_OUTPUT
	Done: BOOL;
	Active: BOOL;
	Error: BOOL;
	ErrorID: ERROR_CODE;
	ErrorIdent: ERROR_STRUCT;
	NbAxis: UDINT;
END_VAR
VAR_IN_OUT
	Axis: ARRAY[*] OF STRING;
END_VAR
VAR
	_browseNode : CXA_DATALAYER.DL_BrowseNode; 
	_diArrayIndex : DINT; 
END_VAR

// example to browse all existing axisprofile 

// call fb, to browse for all configured axisprofile
_browseNode(
	Execute:= Execute, 
	Active=> Active, 
	Error=> Error, 
	ErrorID=> ErrorID, 
	ErrorIdent=> ErrorIdent, 
	NodeName:= 'motion/axs');
	
// check for done
IF _browseNode.Done THEN
	// check, if array size is large enough for the returned 
	IF (UDINT_TO_DINT(_browseNode.ChildNum) > (UPPER_BOUND(Axis, 1)-LOWER_BOUND(Axis, 1))) THEN 
		// array size not large enough => error
		Error:= TRUE;
		ErrorIdent.Table:= USER1_TABLE;
 		ErrorIdent.Additional1:= 16#0E0F0001; 
		ErrorIdent.Additional2:= 16#00000000;  
	ELSE 	
		// array size large enough => assign values
	  	FOR _diArrayIndex:= 0 TO (UPPER_BOUND(Axis, 1)-LOWER_BOUND(Axis, 1)) DO
			Axis[LOWER_BOUND(Axis, 1)+_diArrayIndex]:= _browseNode.GetChildName(Index:= DINT_TO_UDINT(_diArrayIndex));
		END_FOR
		// number of axis
		NbAxis:= _browseNode.ChildNum;
	END_IF
END_IF
// actualise output done
Done:= _browseNode.Done AND NOT Error;

END_FUNCTION_BLOCK

// InternHelpers/MapDriveConnect
FUNCTION_BLOCK MapDriveConnect
VAR_INPUT
	bExecute: BOOL;
END_VAR
VAR_IN_OUT
	instAxisInfoMap: AxisInfoMap;
END_VAR
VAR_OUTPUT
	bDone: BOOL;
	bActive: BOOL;
	bError: BOOL;
	enErrorID: CXA_Datalayer.ERROR_CODE;
	stErrorIdent: CXA_Datalayer.ERROR_STRUCT;
	uiErrorStep: UINT;
END_VAR
VAR
	_DeviceList: iList;
	_GetAllDriveConnectDevices: GetAllDriveConnectDevices;
	_uiState: UINT;
	_uiNextState: UINT;
	_iSubDevice: UINT;
	_stNode: typeDeviceConnectNode;
	_DLReadNodeCtrlx: DL_ReadNode;
	_DLReadNodeIndra: DL_ReadNode;
	_sECatAddrCtrlx: STRING;
	_sReadNodeCtrlx: STRING(255);
	_stAxisInfo: typeAxisInfo;
	_arStrings: ARRAY[0..1] OF POINTER TO STRING(255);
	_sECatAddrIndra: STRING(255);
	_sReadNodeIndra: STRING(255);
	_uiEcat: UDINT;
END_VAR
VAR CONSTANT
	IDLE: UINT := 0;
	GET_DEVICES: UINT := 1;
	MAP_DEVICES: UINT := 2;
	DONE: UINT := 3;
	ERROR: UINT := 4;
	_sEcatAddrNodeCtrlX: STRING := '/sercos-idns/S-0-1042.0.0/data';
	_sEcatAddrNodeIndra: STRING := '/sercos-idns/P-0-4089.0.4/data';
END_VAR

_uiNextState := _uiState; 
CASE _uiState OF 
	IDLE : 
		IF bExecute THEN 
			_uiNextState := GET_DEVICES; 
		END_IF
	GET_DEVICES: 
		IF _GetAllDriveConnectDevices.bError THEN 
			_uiNextState := ERROR; 
			enErrorID := _GetAllDriveConnectDevices.enErrorID; 
			stErrorIdent := _GetAllDriveConnectDevices.stErrorIdent; 
			uiErrorStep := GET_DEVICES; 
		ELSIF _GetAllDriveConnectDevices.bDone THEN 
			IF _DeviceList.GetIterator().Next(ADR(_stNode)) THEN 
				_uiNextState := MAP_DEVICES; 
			ELSE 
				_uiNextState := DONE; 
			END_IF
		END_IF
	MAP_DEVICES: 
		IF _DLReadNodeCtrlx.Error  AND _DLReadNodeIndra.Error THEN 
			_uiNextState := ERROR; 
			enErrorID := _DLReadNodeCtrlx.ErrorID; 
			stErrorIdent := _DLReadNodeCtrlx.ErrorIdent; 
			uiErrorStep := MAP_DEVICES; 
		ELSIF _DLReadNodeCtrlx.Done AND NOT _DLReadNodeCtrlx.Error THEN 
			 _uiEcat := StringHexTOUDINT(_sECatAddrCtrlx); 
		ELSIF _DLReadNodeIndra.Done AND NOT _DLReadNodeIndra.Error THEN 
			 _uiEcat := StrDecToUDINT(_sEcatAddrIndra); 
		END_IF 
		IF  (_DLReadNodeCtrlx.Done AND NOT _DLReadNodeCtrlx.Error) OR (_DLReadNodeIndra.Done AND NOT _DLReadNodeIndra.Error) THEN 
			 IF (instAxisInfoMap.TryGetInfoFromAddr(_uiEcat,stAxisInfo => _stAxisInfo)) THEN  
			 	_stAxisInfo.sDriveConnectName := _stNode.sNodeName; 
				IL_StrSplit(ADR(_stNode.arSubDevices[_iSubDevice]),'-',2,FALSE,ADR(_arStrings),SIZEOF(_arStrings));
			 	_stAxisInfo.iDriveConnectSubDevice := TO_UINT(_arStrings[1]^); 
			 	instAxisInfoMap.TryPutInfo(_stAxisInfo.sAxisName,_stAxisInfo,TRUE);
			 END_IF 
			 _iSubDevice := _iSubdevice + 1; 
			 IF _iSubDevice >= _stNode.uiNumbSubDevices THEN 
				 _iSubDevice := 0; 
				IF _DeviceList.GetIterator().Next(ADR(_stNode))THEN
					_DLReadNodeCtrlx(Execute := FALSE); 
					_DLReadNodeIndra(Execute := FALSE); 
				ELSE 
					 _uiNextState := DONE; 
				END_IF
			 ELSE 
				_DLReadNodeCtrlx(Execute := FALSE); 
				_DLReadNodeIndra(Execute := FALSE);
			 END_IF
		END_IF
		
	DONE, ERROR: 
		IF NOT bExecute THEN 
			_uiNextState := IDLE; 
		END_IF
END_CASE
_uiState := _uiNextState;
CASE _uiState OF 
	IDLE : 
		_iSubDevice := 0; 
	GET_DEVICES: 
		;
	MAP_DEVICES: 
		_sReadNodeCtrlx := 'devices/drives/'; 
		_sReadNodeCtrlx := CONCAT(_sReadNodeCtrlx,_stNode.sNodeName); 
		_sReadNodeCtrlx := CONCAT(_sReadNodeCtrlx,'/subdevices/'); 
		_sReadNodeCtrlx := CONCAT(_sReadNodeCtrlx, _stNode.arSubDevices[_iSubDevice]); 
		_sReadNodeCtrlx := CONCAT(_sReadNodeCtrlx, _sEcatAddrNodeCtrlX); 
		
		_sReadNodeIndra := 'devices/drives/'; 
		_sReadNodeIndra := CONCAT(_sReadNodeIndra,_stNode.sNodeName); 
		_sReadNodeIndra := CONCAT(_sReadNodeIndra,'/subdevices/'); 
		_sReadNodeIndra := CONCAT(_sReadNodeIndra, _stNode.arSubDevices[_iSubDevice]); 
		_sReadNodeIndra := CONCAT(_sReadNodeIndra, _sEcatAddrNodeIndra); 
	DONE, ERROR :
		; 
END_CASE 
_GetAllDriveConnectDevices(bExecute := _uiState = GET_DEVICES, 
						   iDeviceList => _DeviceList); 
_DLReadNodeCtrlx(Execute := _uiState = MAP_DEVICES,
			NodeName := _sReadNodeCtrlx,
			Value := _sECatAddrCtrlx); 
_DLReadNodeIndra(Execute := _uiState = MAP_DEVICES,
			NodeName := _sReadNodeIndra,
			Value := _sECatAddrIndra); 			
bDone := _uiState = DONE; 
bError := _uiState = ERROR; 
bActive := _uiState <> IDLE and _uiState <> ERROR and _uiState <> DONE;

END_FUNCTION_BLOCK

// InternHelpers/StringHexToUDINT
FUNCTION StringHexToUDINT : UDINT
VAR_INPUT
	sHex: STRING(255);
END_VAR
VAR
	_i: INT;
	_multiple: UDINT;
	_decVal: UDINT;
	_byteVal: UDINT;
END_VAR

_multiple := 1; 
FOR _i :=LEN(sHex) - 1 TO 0 BY -1 DO
	_byteVal := sHex[_i]; 
	IF _byteVal >= 48 AND _byteVal <=57 THEN 
		_decVal := _decVal + (_byteVal - 48)* _multiple; 
	ELSIF _byteVal >= 65 AND _byteVal <= 70 THEN 
		_decVal := _decVal + (_byteVal -55) * _multiple; 
	ELSIF _byteVal >= 97 AND _byteVal <= 102 THEN 
		_decVal := _decVal + (_byteVal -87) * _multiple; 
	END_IF
	_multiple := _multiple * 16; 
END_FOR
StringHexToUDINT := _decVal;

END_FUNCTION

// InternHelpers/StringHexToUDINT
{attribute 'hide'}
(*tuns hex string values (as returned by Drive Connect) into a UDIT*) 
FUNCTION StringHexToUDINT : UDINT
VAR_INPUT
	sHex: STRING(255);
END_VAR
VAR
	_i: INT;
	_multiple: UDINT;
	_decVal: UDINT;
	_byteVal: UDINT;
END_VAR

_multiple := 1; 
FOR _i :=LEN(sHex) - 1 TO 0 BY -1 DO
	_byteVal := sHex[_i]; 
	IF _byteVal >= 48 AND _byteVal <=57 THEN 
		_decVal := _decVal + (_byteVal - 48)* _multiple; 
	ELSIF _byteVal >= 65 AND _byteVal <= 70 THEN 
		_decVal := _decVal + (_byteVal -55) * _multiple; 
	ELSIF _byteVal >= 97 AND _byteVal <= 102 THEN 
		_decVal := _decVal + (_byteVal -87) * _multiple; 
	END_IF
	_multiple := _multiple * 16; 
END_FOR
StringHexToUDINT := _decVal;

END_FUNCTION

// InternHelpers/StrDecToUDINT
FUNCTION StrDecToUDINT : UDINT
VAR_INPUT
	sHex: STRING(255);
END_VAR
VAR
	_i: INT;
	_multiple: UDINT;
	_decVal: UDINT;
	_byteVal: UDINT;
END_VAR

_multiple := 1; 
FOR _i :=LEN(sHex) - 1 TO 0 BY -1 DO
	_byteVal := sHex[_i]; 
	IF _byteVal >= 48 AND _byteVal <=57 THEN 
		_decVal := _decVal + (_byteVal - 48)* _multiple; 
	END_IF
	_multiple := _multiple * 10; 
END_FOR
StrDecToUDINT := _decVal;

END_FUNCTION

// InternHelpers/MapDriveConnect
{attribute 'hide'}
(* Maps Drive Connect Data to Axis Data*) 
FUNCTION_BLOCK MapDriveConnect
VAR_INPUT
	bExecute: BOOL;
END_VAR
VAR_IN_OUT
	instAxisInfoMap: AxisInfoMap;
END_VAR
VAR_OUTPUT
	bDone: BOOL;
	bActive: BOOL;
	bError: BOOL;
	enErrorID: CXA_Datalayer.ERROR_CODE;
	stErrorIdent: CXA_Datalayer.ERROR_STRUCT;
	uiErrorStep: UINT;
END_VAR
VAR
	_DeviceList: iList;
	_GetAllDriveConnectDevices: GetAllDriveConnectDevices;
	_uiState: UINT;
	_uiNextState: UINT;
	_iSubDevice: UINT;
	_stNode: typeDeviceConnectNode;
	_DLReadNode: DL_ReadNode;
	_sECatAddr: STRING;
	_sReadNode: STRING(255);
	_stAxisInfo: typeAxisInfo;
	_arStrings: ARRAY[0..1] OF POINTER TO STRING(255);
END_VAR
VAR CONSTANT
	IDLE: UINT := 0;
	GET_DEVICES: UINT := 1;
	MAP_DEVICES: UINT := 2;
	DONE: UINT := 3;
	ERROR: UINT := 4;
	_sEcatAddrNode: STRING := '/sercos-idns/S-0-1042.0.0/data';
END_VAR

_uiNextState := _uiState; 
CASE _uiState OF 
	IDLE : 
		IF bExecute THEN 
			_uiNextState := GET_DEVICES; 
		END_IF
	GET_DEVICES: 
		IF _GetAllDriveConnectDevices.bError THEN 
			_uiNextState := ERROR; 
			enErrorID := _GetAllDriveConnectDevices.enErrorID; 
			stErrorIdent := _GetAllDriveConnectDevices.stErrorIdent; 
			uiErrorStep := GET_DEVICES; 
		ELSIF _GetAllDriveConnectDevices.bDone THEN 
			IF _DeviceList.GetIterator().Next(ADR(_stNode)) THEN 
				_uiNextState := MAP_DEVICES; 
			ELSE 
				_uiNextState := DONE; 
			END_IF
		END_IF
	MAP_DEVICES: 
		IF _DLReadNode.Error THEN 
			_uiNextState := ERROR; 
			enErrorID := _DLReadNode.ErrorID; 
			stErrorIdent := _DLReadNode.ErrorIdent; 
			uiErrorStep := MAP_DEVICES; 
		ELSIF _DLReadNode.Done THEN  
			 IF (instAxisInfoMap.TryGetInfoFromAddr(StringHexTOUDINT(_sEcatAddr),stAxisInfo => _stAxisInfo)) THEN  
			 	_stAxisInfo.sDriveConnectName := _stNode.sNodeName; 
				IL_StrSplit(ADR(_stNode.arSubDevices[_iSubDevice]),'-',2,FALSE,ADR(_arStrings),SIZEOF(_arStrings));
			 	_stAxisInfo.iDriveConnectSubDevice := TO_UINT(_arStrings[1]^); 
			 	instAxisInfoMap.TryPutInfo(_stAxisInfo.sAxisName,_stAxisInfo);
			 END_IF 
			 _iSubDevice := _iSubdevice + 1; 
			 IF _iSubDevice >= _stNode.uiNumbSubDevices THEN 
				 _iSubDevice := 0; 
				IF _DeviceList.GetIterator().Next(ADR(_stNode))THEN
					_DLreadNode(Execute := FALSE); 
				ELSE 
					 _uiNextState := DONE; 
				END_IF
			 ELSE 
				_DLreadNode(Execute := FALSE); 
			 END_IF
		END_IF
	DONE, ERROR: 
		IF NOT bExecute THEN 
			_uiNextState := IDLE; 
		END_IF
END_CASE
_uiState := _uiNextState;
CASE _uiState OF 
	IDLE : 
		_iSubDevice := 0; 
	GET_DEVICES: 
		;
	MAP_DEVICES: 
		_sReadNode := 'devices/drives/'; 
		_sReadNode := CONCAT(_sReadNode,_stNode.sNodeName); 
		_sReadNode := CONCAT(_sReadNode,'/subdevices/'); 
		_sReadNode := CONCAT(_sReadNode, _stNode.arSubDevices[_iSubDevice]); 
		_sReadNode := CONCAT(_sReadNode, _sEcatAddrNode); 
	DONE, ERROR :
		; 
END_CASE 
_GetAllDriveConnectDevices(bExecute := _uiState = GET_DEVICES, 
						   iDeviceList => _DeviceList); 
_DLReadNode(Execute := _uiState = MAP_DEVICES,
			NodeName := _sReadNode,
			Value := _sECatAddr); 
			
bDone := _uiState = DONE; 
bError := _uiState = ERROR; 
bActive := _uiState <> IDLE and _uiState <> ERROR and _uiState <> DONE;

END_FUNCTION_BLOCK

// InternHelpers/GetAllDriveConnectDevices
FUNCTION_BLOCK GetAllDriveConnectDevices
VAR_INPUT
	bExecute: BOOL;
END_VAR
VAR_OUTPUT
	bDone: BOOL;
	bError: BOOL;
	iDeviceList: iList;
	uiErrorStep: UINT;
	enErrorID: CXA_Datalayer.ERROR_CODE;
	stErrorIdent: CXA_Datalayer.ERROR_STRUCT;
END_VAR
VAR
	DeviceConnectNodes: DeviceConnectNodeContainer;
	DeviceConnectList: List := (DataContainer := DeviceConnectNodes);
	_stDeviceNode: typeDeviceConnectNode;
	_uiState: UINT;
	_uiNextState: UINT;
	_DLBrowseDevices: CXA_DATALAYER.DL_BrowseNode;
	_DLBrowseSubDevices: CXA_DATALAYER.DL_BrowseNode;
	_iDevice: INT;
	_sBrowseSubDeviceString: STRING(255);
	_sBrowseDevices: STRING(255) := 'devices/drives';
	_i: UDINT;
END_VAR
VAR CONSTANT
	IDLE: UINT := 0;
	BROWSE_DEVICES: UINT := 1;
	BROWSE_SUB_DEVICES: UINT := 2;
	DONE: UINT := 3;
	ERROR: UINT := 4;
END_VAR

_uiNextState := _uiState; 
CASE _uiState OF 
	IDLE: 
		IF bExecute THEN 
			_uiNextState := BROWSE_DEVICES; 
		END_IF
	BROWSE_DEVICES: 
		IF _DLBrowseDevices.Error THEN 
			_uiNextState := ERROR; 
			stErrorIdent := _DLBrowseDevices.ErrorIdent; 
			enErrorID    := _DLBrowseDevices.ErrorID; 
			uiErrorStep := BROWSE_DEVICES; 
		ELSIF _DLBrowseDevices.Done THEN 
			IF _DLBrowseDevices.ChildPtr = 0 THEN 
				_uiNextState := ERROR; 
				uiErrorStep := BROWSE_DEVICES;
			ELSE 
				_uiNextState := BROWSE_SUB_DEVICES; 
			END_IF
		END_IF
	BROWSE_SUB_DEVICES: 
		IF _dlBrowseSubDevices.Error THEN 
			_uiNextState := ERROR; 
			stErrorIdent := _DLBrowseSubDevices.ErrorIdent; 
			enErrorID    := _DLBrowseSubDevices.ErrorID; 
			uiErrorStep := BROWSE_SUB_DEVICES; 
		ELSIF _dlBrowseSubDevices.Done THEN 
			IF _dlBrowseSubDevices.ChildPtr = 0 THEN 
				_uiState := ERROR; 
				uiErrorStep := BROWSE_SUB_DEVICES;
			ELSE
				_stDeviceNode.sNodeName := _dlBrowseDevices.ChildPtr[_iDevice]^; 
				FOR _i := 0 TO _DLBrowseSubDevices.ChildNum - 1 DO 
					_stDeviceNode.arSubDevices[_i] := _DLBrowseSubDevices.ChildPtr[_i]^; 
				END_FOR
				_stDeviceNode.uiNumbSubDevices := TO_UINT(_i); 
				DeviceConnectList.PushBack(ADR(_stDeviceNode)); 
				_iDevice := _iDevice + 1; 
				IF _iDevice > TO_DINT(_DLBrowseDevices.ChildNum) - 1 THEN 
					_uiNextState := DONE; 
				ELSE 
					_dlBrowseSubDevices(Execute := FALSE); 
				END_IF
			END_IF
		END_IF
	DONE, ERROR: 
		IF NOT bExecute THEN 
			_uiNextState := IDLE; 
		END_IF
END_CASE
_uiState := _uiNextState; 
CASE _uiState OF 
	IDLE: 
		_iDevice := 0; 
		uiErrorStep := 0; 
		enErrorID := CXA_Datalayer.ERROR_CODE.NONE_ERROR; 
	BROWSE_DEVICES: 
		DeviceConnectList.Clear();
	BROWSE_SUB_DEVICES: 
		_sBrowseSubDeviceString := Concat(_sBrowseDevices,'/');
		_sBrowseSubDeviceString := Concat(_sBrowseSubDeviceString, _DLBrowseDevices.ChildPtr[_iDevice]^); 
		_sBrowseSubDeviceString := Concat(_sBrowseSubDeviceString, '/subdevices'); 
	DONE, ERROR: 
		;
END_CASE
_DLBrowseDevices(Execute := _uiState = BROWSE_DEVICES,
				 NodeName := _sBrowseDevices); 
_DLBrowseSubDevices(Execute := _uiState = BROWSE_SUB_DEVICES, 
					NodeName := _sBrowseSubDeviceString); 
iDeviceList := DeviceConnectList; 
bDone := _uiState = DONE; 
bError := _uiState = ERROR;

END_FUNCTION_BLOCK

// InternHelpers/GetAllDriveConnectDevices
{attribute 'hide'}
(*Iterates thru drive connect devices getting info needed to map them*) 
FUNCTION_BLOCK GetAllDriveConnectDevices
VAR_INPUT
	bExecute: BOOL;
END_VAR
VAR_OUTPUT
	bDone: BOOL;
	bError: BOOL;
	iDeviceList: iList;
	uiErrorStep: UINT;
	enErrorID: CXA_Datalayer.ERROR_CODE;
	stErrorIdent: CXA_Datalayer.ERROR_STRUCT;
END_VAR
VAR
	DeviceConnectNodes: DeviceConnectNodeContainer;
	DeviceConnectList: List := (DataContainer := DeviceConnectNodes);
	_stDeviceNode: typeDeviceConnectNode;
	_uiState: UINT;
	_uiNextState: UINT;
	_DLBrowseDevices: CXA_DATALAYER.DL_BrowseNode;
	_DLBrowseSubDevices: CXA_DATALAYER.DL_BrowseNode;
	_iDevice: INT;
	_sBrowseSubDeviceString: STRING(255);
	_sBrowseDevices: STRING(255) := 'devices/drives';
	_i: UDINT;
END_VAR
VAR CONSTANT
	IDLE: UINT := 0;
	BROWSE_DEVICES: UINT := 1;
	BROWSE_SUB_DEVICES: UINT := 2;
	DONE: UINT := 3;
	ERROR: UINT := 4;
END_VAR

_uiNextState := _uiState; 
CASE _uiState OF 
	IDLE: 
		IF bExecute THEN 
			_uiNextState := BROWSE_DEVICES; 
		END_IF
	BROWSE_DEVICES: 
		IF _DLBrowseDevices.Error THEN 
			_uiNextState := ERROR; 
			stErrorIdent := _DLBrowseDevices.ErrorIdent; 
			enErrorID    := _DLBrowseDevices.ErrorID; 
			uiErrorStep := BROWSE_DEVICES; 
		ELSIF _DLBrowseDevices.Done THEN 
			_uiNextState := BROWSE_SUB_DEVICES; 
		END_IF
	BROWSE_SUB_DEVICES: 
		IF _dlBrowseSubDevices.Error THEN 
			_uiNextState := ERROR; 
			stErrorIdent := _DLBrowseSubDevices.ErrorIdent; 
			enErrorID    := _DLBrowseSubDevices.ErrorID; 
			uiErrorStep := BROWSE_SUB_DEVICES; 
		ELSIF _dlBrowseSubDevices.Done THEN 
			_stDeviceNode.sNodeName := _dlBrowseDevices.ChildPtr[_iDevice]^; 
			FOR _i := 0 TO _DLBrowseSubDevices.ChildNum - 1 DO 
				_stDeviceNode.arSubDevices[_i] := _DLBrowseSubDevices.ChildPtr[_i]^; 
			END_FOR
			_stDeviceNode.uiNumbSubDevices := TO_UINT(_i); 
			DeviceConnectList.PushBack(ADR(_stDeviceNode)); 
			_iDevice := _iDevice + 1; 
			IF _iDevice > TO_DINT(_DLBrowseDevices.ChildNum) - 1 THEN 
				_uiNextState := DONE; 
			ELSE 
				_dlBrowseSubDevices(Execute := FALSE); 
			END_IF
		END_IF
	DONE, ERROR: 
		IF NOT bExecute THEN 
			_uiNextState := IDLE; 
		END_IF
END_CASE
_uiState := _uiNextState; 
CASE _uiState OF 
	IDLE: 
		_iDevice := 0; 
		uiErrorStep := 0; 
		enErrorID := CXA_Datalayer.ERROR_CODE.NONE_ERROR; 
	BROWSE_DEVICES: 
		;
	BROWSE_SUB_DEVICES: 
		_sBrowseSubDeviceString := Concat(_sBrowseDevices,'/');
		_sBrowseSubDeviceString := Concat(_sBrowseSubDeviceString, _DLBrowseDevices.ChildPtr[_iDevice]^); 
		_sBrowseSubDeviceString := Concat(_sBrowseSubDeviceString, '/subdevices'); 
	DONE, ERROR: 
		;
END_CASE
_DLBrowseDevices(Execute := _uiState = BROWSE_DEVICES,
				 NodeName := _sBrowseDevices); 
_DLBrowseSubDevices(Execute := _uiState = BROWSE_SUB_DEVICES, 
					NodeName := _sBrowseSubDeviceString); 
iDeviceList := DeviceConnectList; 
bDone := _uiState = DONE; 
bError := _uiState = ERROR;

END_FUNCTION_BLOCK

// InternHelpers/Containers/DeviceConnectNodeContainer
{attribute 'no_check' := ''}
FUNCTION_BLOCK DeviceConnectNodeContainer IMPLEMENTS iDataContainer
{attribute 'hide'}
VAR CONSTANT
	_size : UDINT := Param.MAX_AXIS;
END_VAR 
VAR
	_arBacking: ARRAY[0.._size -1] OF typeDeviceConnectNode;
	_pData: POINTER TO typeDeviceConnectNode;
END_VAR

{attribute 'hide'}
{attribute 'no_check' := ''}
METHOD Get : BOOL
VAR_INPUT
	index: UDINT;
	pData: PVoid;
END_VAR
_pData := pData; 
IF index < _size THEN 
	_pData^ := _arBacking[index]; 
	Get := TRUE;
ELSE 
	Get := FALSE; 
END_IF
END_METHOD

{attribute 'hide'}
{attribute 'no_check' := ''}
METHOD GetPointer : PVoid
VAR_INPUT
	index: UDINT;
END_VAR
IF index < _size THEN 
	GetPointer:= ADR(_arBacking[index]); 
ELSE 
	GetPointer := 0; 
END_IF
END_METHOD

{attribute 'hide'}
METHOD GetSize : UDINT
GetSize := _size;
END_METHOD

{attribute 'hide'}
{attribute 'no_check' := ''}
METHOD Put : BOOL
VAR_INPUT
	index: UDINT;
	pData: PVoid;
END_VAR
_pData := pData; 
IF index < _size THEN 
	_arBacking[index] := _pData^; 
	Put := TRUE; 
ELSE 
	Put := FALSE; 
END_IF
END_METHOD

END_FUNCTION_BLOCK

// InternHelpers/Containers/DeviceConnectNodeContainer
{attribute 'no_check' := ''}
FUNCTION_BLOCK DeviceConnectNodeContainer IMPLEMENTS iDataContainer
VAR CONSTANT
	_size: UDINT := Param.MAX_AXIS;
END_VAR
VAR
	_arBacking: ARRAY[0..(_size - 1)] OF typeDeviceConnectNode;
	_pData: POINTER TO typeDeviceConnectNode;
END_VAR

END_FUNCTION_BLOCK

// DriveParamBackup
FUNCTION_BLOCK DriveParamBackup
VAR_INPUT
	bExecute: BOOL;
	bOverwrite: BOOL;
	sDriveConnectName: STRING;
	iSubDevice: UINT;
	sFileName: STRING;
	enBackupType: comm_drive_ExportParFile_ParametersType;
END_VAR
VAR_OUTPUT
	bDone: BOOL;
	bActive: BOOL;
	bError: BOOL;
	uiProgress: UDINT;
	enTaskState: comm_datalayer_ProgramTaskState;
	ErrorCause: EN_DRIVE_BACKUP_RESTORE_ERROR;
	ErrorID: CXA_Datalayer.ERROR_CODE;
	ErrorIdent: CXA_Datalayer.ERROR_STRUCT;
	sFailureInfo: STRING;
END_VAR
VAR
	_builder: Flatbuffers.FlatBufferBuilder;
	_backUpReq: comm_drive_ExportParFile_ExportParFile;
	_taskStatus: comm_Datalayer_ProgramTask;
	_pRespString: POINTER TO STRING(255);
	_sRespString: STRING(255);
	_dlCreateNode: CXA_DataLayer.DL_CreateNodeValue;
	_dlReadNode: CXA_DataLayer.DL_ReadNodeValue;
	_dlBackupReq: CXA_DataLayer.DL_NodeValue;
	_dlTaskPath: CXA_DataLayer.DL_NodeValue;
	_dlTaskResp: CXA_Datalayer.DL_NodeValue;
	_uiState: UINT;
	_uiNextState: UINT;
	_enTaskState: comm_datalayer_ProgramTaskState;
	_sReqString: STRING(255);
	_sSaveString: STRING(255);
	_uiOffset: UDINT;
	_browseForFile: DCBrowseForFile;
	_dlDeleteNode: CXA_DataLayer.DL_DeleteNode;
	_sDeleteNode: STRING(255);
END_VAR
VAR CONSTANT
	STATE_IDLE: UINT := 0;
	STATE_FIND_FILE: UINT := 1;
	STATE_DELETE_FILE: UINT := 2;
	STATE_REQ: UINT := 3;
	STATE_BACKING_UP: UINT := 4;
	STATE_DONE: UINT := 5;
	STATE_ERROR: UINT := 6;
	S_PATH_DEVICES: STRING := 'devices/drives/';
	S_PATH_BACKUPS: STRING := 'filesystem/parameterfiles/';
END_VAR

CASE _uiState OF 
	STATE_IDLE: 
		IF bExecute THEN 
			_uiNextState := STATE_FIND_FILE; 
		END_IF
	STATE_FIND_FILE: 
		IF _browseForFile.bError THEN 
			ErrorID := _browseForFile.ErrorID; 
			ErrorIdent := _browseForFile.ErrorIdent; 
			ErrorCause :=EN_DRIVE_BACKUP_RESTORE_ERROR.FileBrowseFailed; 
			_uiNextState := STATE_ERROR; 
		ELSIF _browseForFile.bDone THEN 
			IF _browseForFile.bFound AND NOT bOverwrite THEN 
				ErrorCause := EN_DRIVE_BACKUP_RESTORE_ERROR.FileExists; 
				_uiNextState := STATE_ERROR; 
			ELSIF _browseForFile.bFound THEN 
				_uiNextState := STATE_DELETE_FILE; 
			ELSE 
				_uiNextState := STATE_REQ; 
			END_IF;  
		END_IF
	STATE_DELETE_FILE: 
		IF _dlDeleteNode.Error THEN 
			ErrorID := _dlDeleteNode.ErrorID; 
			ErrorIdent := _dlDeleteNode.ErrorIdent; 
			ErrorCause := EN_DRIVE_BACKUP_RESTORE_ERROR.DeleteFailed; 
		ELSIF _dlDeleteNode.Done THEN 
			_uiNextState := STATE_REQ; 
		END_IF
	STATE_REQ: 
		IF _dlCreateNode.Error THEN 
			_uiNExtState := STATE_ERROR; 
			ErrorID := _dlCreateNode.ErrorID;
			ErrorIDent := _dlCreateNode.ErrorIdent; 
			ErrorCause := EN_DRIVE_BACKUP_RESTORE_ERROR.RequestFailed;  
		ELSIF _dlCreateNode.Done THEN 
			_uiNextState := STATE_BACKING_UP; 
		END_IF
	STATE_BACKING_UP: 
		IF _dlReadNode.Error THEN 
			_uiNextState := STATE_ERROR; 
			ErrorID := _dlReadNode.ErrorID;
			ErrorIDent := _dlReadNode.ErrorIdent; 
			ErrorCause := EN_DRIVE_BACKUP_RESTORE_ERROR.ProgressReadFailed;  
		ELSIF _dlReadNode.Done THEN 
			IF _enTaskState = comm_datalayer_ProgramTaskState.failed THEN 
				_uiNextState := STATE_ERROR; 
				ErrorID := _dlReadNode.ErrorID;
				ErrorIdent := _dlReadNode.ErrorIdent; 
				ErrorCause := EN_DRIVE_BACKUP_RESTORE_ERROR.BackupFailed;  
				sFailureInfo := _taskStatus.getProgressInfo(); 
			ELSIF _enTaskState = comm_datalayer_ProgramTaskState.done THEN 
				_uiNextState := STATE_DONE; 
			ELSE
				_dlReadNode(Execute := FALSE); 
			END_IF
		END_IF
	STATE_DONE, STATE_ERROR: 
		IF NOT bExecute THEN 
			_uiNextState := STATE_IDLE; 
		END_IF
END_CASE
_uiState := _uiNextState; 
CASE _uiState OF 
	STATE_IDLE: 
		_dlReadNode.Execute := FALSE; 
		_dlCreateNode.Execute := FALSE; 
		_browseForFile.bExecute := FALSE; 
		_dlDeleteNode.Execute := FALSE; 
		sFailureInfo := 'OK'; 
		enTaskState := comm_datalayer_ProgramTaskState.done; 
		ErrorCause := EN_DRIVE_BACKUP_RESTORE_ERROR.OK; 
		uiProgress := 0; 
		
	STATE_FIND_FILE: 
		_browseForFile.sFileName := sFileName; 
		_browseForFile.bExecute := TRUE; 
		
	STATE_DELETE_FILE: 
		_dlDeleteNode.Execute := TRUE; 
		_sDeleteNode :='driveconnect/'; 
		_sDeleteNode := Concat(_sDeleteNode,S_PATH_BACKUPS);
		_sDeleteNode := Concat(_sDeleteNode,sFileName); 
		
	STATE_REQ: 
		_dlCreateNode.Execute := TRUE; 
		_builder(forceDefaults := TRUE); 
		_sSaveString := CONCAT(S_PATH_BACKUPS,sFileName); 
		_sReqString := CONCAT(S_PATH_DEVICES,sDriveConnectName); 
		_sReqString := CONCAT(_sReqString,'/subdevices/subdevice-'); 
		_sReqString := CONCAT(_sReqString,INT_TO_STRING(iSubDevice)); 
		_sReqString := CONCAT(_sReqString,'/export-parameter'); 
		_uiOffset := _backUpReq.createExportParFile(_builder,_sSaveString,enBackupType);
 		_builder.finish(_uiOffset); 
		_dlBackupReq.SetFlatbuffer(_builder); 
	STATE_BACKING_UP: 
		_pRespString := _dlTaskPath.GetData(); 
		_sRespString := _pRespString^; 
		_dlReadNode.Execute := TRUE; 
END_CASE

_dlCreateNode(NodeName := _sReqString,
			  NodeValueIn := _dlBackupReq, 
			  NodeValueOut := _dlTaskPath); 
			  
_dlReadNode(NodeName := _sRespString,
			NodeValue := _dlTaskResp); 
			
_browseForFile(); 

_dlDeleteNode(NodeName := _sDeleteNode); 

IF _dlReadNode.Done THEN 
	_taskStatus.getRootAsProgramTask(_dlTaskResp.GetData(),_dlTaskResp.GetSize()); 
	_enTaskState := _taskStatus.getState(); 
	uiProgress := _taskStatus.getProgress(); 
	enTaskState := _enTaskState; 
END_IF

bActive := _uiState <> STATE_IDLE AND _uiState <> STATE_DONE AND _uiState <> STATE_ERROR; 
bDone := _uiState = STATE_DONE; 
bError := _uiState = STATE_ERROR;

END_FUNCTION_BLOCK

// InternHelpers/comm_drive_ExportParFile_ExportParFile
///automatically generated by the FlatBuffers compiler, do not modify
///comm\drive\ExportParFile
///Import FlatBuffers Library
FUNCTION_BLOCK comm_drive_ExportParFile_ExportParFile EXTENDS flatbuffers.Table
VAR
	_builder: REFERENCE TO flatbuffers.FlatBufferBuilder;
	_bb: flatbuffers.ByteBuffer;
END_VAR

///automatically generated by the FlatBuffers compiler, do not modify
///comm\drive\ExportParFile
///
///Set the values of a ExportParFile and return it.
{attribute 'conditionalshow' := ''}
METHOD _assign : comm_drive_ExportParFile_ExportParFile
VAR_INPUT
	i: UDINT;
	_bb: REFERENCE TO flatbuffers.ByteBuffer;
END_VAR
_init(i:=i, _bb:=_bb);
_assign:=this^;
END_METHOD

///automatically generated by the FlatBuffers compiler, do not modify
///comm\drive\ExportParFile
///
///Set the values of a table.
{attribute 'conditionalshow' := ''}
METHOD _init
VAR_INPUT
	i: UDINT;
	_bb: REFERENCE TO flatbuffers.ByteBuffer;
END_VAR
_reset(i:=i, _bb:=_bb);
END_METHOD

///automatically generated by the FlatBuffers compiler, do not modify
///comm\drive\ExportParFile
///
///Add values to the table.
METHOD addBackupType
VAR_INPUT
	backupType: comm_drive_ExportParFile_ParametersType;
END_VAR
IF NOT __ISVALIDREF(_builder) THEN
  SysExceptGenerateException(RTSEXCPT_INVALID_HANDLE);
END_IF
_builder.add_UDINT(o:=1, x:=backupType, d:=0);
END_METHOD

///automatically generated by the FlatBuffers compiler, do not modify
///comm\drive\ExportParFile
///
///Add values to the table.
METHOD addFileName
VAR_INPUT
	fileNameOffset: UDINT;
END_VAR
IF NOT __ISVALIDREF(_builder) THEN
  SysExceptGenerateException(RTSEXCPT_INVALID_HANDLE);
END_IF
_builder.add_Offset(o:=0, x:=fileNameOffset, d:=0);
END_METHOD

///automatically generated by the FlatBuffers compiler, do not modify
///comm\drive\ExportParFile
///
///Creates a table in the Flatbuffer and returns the offset to it.
METHOD createExportParFile : UDINT
VAR_INPUT
	builder: REFERENCE TO flatbuffers.FlatBufferBuilder;
	fileName: STRING;
	backupType: comm_drive_ExportParFile_ParametersType;
END_VAR
VAR
	fileNameOffset: UDINT;
END_VAR
_builder REF= builder;
IF NOT __ISVALIDREF(_builder) THEN
  SysExceptGenerateException(RTSEXCPT_INVALID_HANDLE);
END_IF
fileNameOffset := builder.createString(fileName);
_builder.startTable(numfields:=2);
addFileName(fileNameOffset:=fileNameOffset);
addBackupType(backupType:=backupType);
createExportParFile := endExportParFile();
END_METHOD

///automatically generated by the FlatBuffers compiler, do not modify
///comm\drive\ExportParFile
///
///End the table and return a offset to it
METHOD endExportParFile : UDINT
VAR
	o: UDINT;
END_VAR
o := _builder.endTable();
_builder REF= 0;
endExportParFile := o;
END_METHOD

///automatically generated by the FlatBuffers compiler, do not modify
///comm\drive\ExportParFile
///
///Returns a UDINT from the table.
METHOD getBackupType : comm_drive_ExportParFile_ParametersType
VAR
	o: UDINT;
END_VAR
o := _offset(vtable_offset:=6);
IF o<>0 THEN
    getBackupType := bb.getUDINT(offset:=o+bb_pos);
ELSE
    getBackupType := 0;
END_IF
END_METHOD

///automatically generated by the FlatBuffers compiler, do not modify
///comm\drive\ExportParFile
///
///Returns a String.
METHOD getFileName : STRING
VAR
	o: UDINT;
END_VAR
o := _offset(vtable_offset:=4);
IF o<>0 THEN
    getFileName := _string(offset:=o+bb_pos);
ELSE
    getFileName := '';
END_IF
END_METHOD

///automatically generated by the FlatBuffers compiler, do not modify
///comm\drive\ExportParFile
///
///Returns a String as pointer to byte.
METHOD getFileNameAsBytePtr : POINTER TO BYTE
VAR
	o: UDINT;
END_VAR
o := _offset(vtable_offset:=4);
IF o<>0 THEN
    getFileNameAsBytePtr := _stringPtr(offset:=o+bb_pos);
ELSE
    getFileNameAsBytePtr := 0;
END_IF
END_METHOD

///automatically generated by the FlatBuffers compiler, do not modify
///comm\drive\ExportParFile
///
///Returns a ExportParFile from the ByteBuffer.
/// 
METHOD getRootAsExportParFile : comm_drive_ExportParFile_ExportParFile
VAR_INPUT
	data: POINTER TO BYTE;
	size: __UXINT;
END_VAR
_bb(data:=data, _capacity:=TO_UDINT(size));
bb REF= _bb;
getRootAsExportParFile := _assign(i:=bb.getUDINT(0), _bb:=bb);
END_METHOD

///automatically generated by the FlatBuffers compiler, do not modify
///comm\drive\ExportParFile
///
///Start the table to add values.
METHOD startExportParFile
VAR_INPUT
	builder: REFERENCE TO flatbuffers.FlatBufferBuilder;
END_VAR
_builder REF= builder;
_builder.startTable(numfields:=2);
END_METHOD

///automatically generated by the FlatBuffers compiler, do not modify
///comm\drive\ExportParFile
METHOD verify : BOOL
VAR_INPUT
	data: POINTER TO BYTE;
	size: __UXINT;
END_VAR
VAR
	_bb: ByteBuffer;
END_VAR
_bb(data:=data, _capacity:=TO_UDINT(size));
verify := verifyExportParFile(data, size, _bb.getUDINT(0));
END_METHOD

///automatically generated by the FlatBuffers compiler, do not modify
///comm\drive\ExportParFile
{attribute 'conditionalshow' := ''}
METHOD verifyExportParFile : BOOL
VAR_INPUT
	data: POINTER TO BYTE;
	size: __UXINT;
	pointer_: UDINT;
END_VAR
VAR
	_bb: ByteBuffer;
	verifier: flatbuffers.Verifier;
	vt_start: UDINT;
	vt_size: UDINT;
END_VAR
_bb(data:=data, _capacity:=TO_UDINT(size));
IF pointer_ = 0 THEN
    verifyExportParFile := TRUE;
    RETURN;
END_IF

if pointer_ > (size - SIZEOF(UDINT)) then
    verifyExportParFile := FALSE;
    return;
END_IF

vt_start := _bb.getUDINT(pointer_);
if (pointer_ - vt_start) > (size - SIZEOF(UDINT)) then
    verifyExportParFile := FALSE;
    return;
END_IF

vt_size := _bb.getUINT(pointer_ - vt_start);
verifier(data:=data, size:=size, pointer_:=pointer_, v_size:=vt_size);

IF verifier.verifyTable() AND verifier.verifyString(4) AND verifier.verifyScalar(6) THEN
    verifyExportParFile := TRUE;
ELSE
    verifyExportParFile := FALSE;
END_IF
END_METHOD

END_FUNCTION_BLOCK

// InternHelpers/comm_datalayer_ProgramTask
///automatically generated by the FlatBuffers compiler, do not modify
///comm\datalayer
///Import FlatBuffers Library
FUNCTION_BLOCK comm_datalayer_ProgramTask EXTENDS flatbuffers.Table
VAR
	_builder: REFERENCE TO flatbuffers.FlatBufferBuilder;
	result1: comm_datalayer_Diagnosis;
	_bb: flatbuffers.ByteBuffer;
END_VAR

///automatically generated by the FlatBuffers compiler, do not modify
///comm\datalayer
///
///Set the values of a ProgramTask and return it.
{attribute 'conditionalshow' := ''}
METHOD _assign : comm_datalayer_ProgramTask
VAR_INPUT
	i: UDINT;
	_bb: REFERENCE TO flatbuffers.ByteBuffer;
END_VAR
_init(i:=i, _bb:=_bb);
_assign:=this^;
END_METHOD

///automatically generated by the FlatBuffers compiler, do not modify
///comm\datalayer
///
///Set the values of a table.
{attribute 'conditionalshow' := ''}
METHOD _init
VAR_INPUT
	i: UDINT;
	_bb: REFERENCE TO flatbuffers.ByteBuffer;
END_VAR
_reset(i:=i, _bb:=_bb);
END_METHOD

///automatically generated by the FlatBuffers compiler, do not modify
///comm\datalayer
///
///Add values to the table.
METHOD addId
VAR_INPUT
	idOffset: UDINT;
END_VAR
IF NOT __ISVALIDREF(_builder) THEN
  SysExceptGenerateException(RTSEXCPT_INVALID_HANDLE);
END_IF
_builder.add_Offset(o:=0, x:=idOffset, d:=0);
END_METHOD

///automatically generated by the FlatBuffers compiler, do not modify
///comm\datalayer
///
///Add values to the table.
METHOD addProgress
VAR_INPUT
	progress: UDINT;
END_VAR
IF NOT __ISVALIDREF(_builder) THEN
  SysExceptGenerateException(RTSEXCPT_INVALID_HANDLE);
END_IF
_builder.add_UDINT(o:=2, x:=progress, d:=0);
END_METHOD

///automatically generated by the FlatBuffers compiler, do not modify
///comm\datalayer
///
///Add values to the table.
METHOD addProgressData
VAR_INPUT
	progressDataOffset: UDINT;
END_VAR
IF NOT __ISVALIDREF(_builder) THEN
  SysExceptGenerateException(RTSEXCPT_INVALID_HANDLE);
END_IF
_builder.add_Offset(o:=5, x:=progressDataOffset, d:=0);
END_METHOD

///automatically generated by the FlatBuffers compiler, do not modify
///comm\datalayer
///
///Add values to the table.
METHOD addProgressInfo
VAR_INPUT
	progressInfoOffset: UDINT;
END_VAR
IF NOT __ISVALIDREF(_builder) THEN
  SysExceptGenerateException(RTSEXCPT_INVALID_HANDLE);
END_IF
_builder.add_Offset(o:=4, x:=progressInfoOffset, d:=0);
END_METHOD

///automatically generated by the FlatBuffers compiler, do not modify
///comm\datalayer
///
///Add values to the table.
METHOD addResult
VAR_INPUT
	resultOffset: UDINT;
END_VAR
IF NOT __ISVALIDREF(_builder) THEN
  SysExceptGenerateException(RTSEXCPT_INVALID_HANDLE);
END_IF
_builder.add_Offset(o:=3, x:=resultOffset, d:=0);
END_METHOD

///automatically generated by the FlatBuffers compiler, do not modify
///comm\datalayer
///
///Add values to the table.
METHOD addState
VAR_INPUT
	state: comm_datalayer_ProgramTaskState;
END_VAR
IF NOT __ISVALIDREF(_builder) THEN
  SysExceptGenerateException(RTSEXCPT_INVALID_HANDLE);
END_IF
_builder.add_BYTE(o:=1, x:=state, d:=0);
END_METHOD

///automatically generated by the FlatBuffers compiler, do not modify
///comm\datalayer
///
///Creates a table in the Flatbuffer and returns the offset to it.
METHOD createProgramTask : UDINT
VAR_INPUT
	builder: REFERENCE TO flatbuffers.FlatBufferBuilder;
	id: STRING;
	/// id of the task
	state: comm_datalayer_ProgramTaskState;
	/// state of the task
	progress: UDINT;
	/// Progress of the task in percent, if it's not possible to calculate, set state to running and progress to 0
	resultOffset: UDINT;
	/// result of task;
	progressInfo: STRING;
	/// Additional progress information
	progressDataOffset: UDINT;
END_VAR
VAR
	idOffset: UDINT;
	progressInfoOffset: UDINT;
END_VAR
_builder REF= builder;
IF NOT __ISVALIDREF(_builder) THEN
  SysExceptGenerateException(RTSEXCPT_INVALID_HANDLE);
END_IF
idOffset := builder.createString(id);
progressInfoOffset := builder.createString(progressInfo);
_builder.startTable(numfields:=6);
addId(idOffset:=idOffset);
addState(state:=state);
addProgress(progress:=progress);
addResult(resultOffset:=resultOffset);
addProgressInfo(progressInfoOffset:=progressInfoOffset);
addProgressData(progressDataOffset:=progressDataOffset);
createProgramTask := endProgramTask();
END_METHOD

///automatically generated by the FlatBuffers compiler, do not modify
///comm\datalayer
METHOD createSortedprogressDataVector : UDINT
VAR_INPUT
	builder: REFERENCE TO flatbuffers.Flatbufferbuilder;
	obj1: REFERENCE TO comm_datalayer_ProgressData;
	offsets: POINTER TO DINT;
	size: UDINT;
END_VAR
createSortedprogressDataVector := builder.createSortedVectorOfTables(bb_:=builder.dataBuffer(), obj:=obj1, offsets := offsets, size:=size);
END_METHOD

///automatically generated by the FlatBuffers compiler, do not modify
///comm\datalayer
///
///End the table and return a offset to it
METHOD endProgramTask : UDINT
VAR
	o: UDINT;
END_VAR
o := _builder.endTable();
_builder REF= 0;
endProgramTask := o;
END_METHOD

///automatically generated by the FlatBuffers compiler, do not modify
///comm\datalayer
///
///Returns a String.
METHOD getId : STRING
VAR
	o: UDINT;
END_VAR
o := _offset(vtable_offset:=4);
IF o<>0 THEN
    getId := _string(offset:=o+bb_pos);
ELSE
    getId := '';
END_IF
END_METHOD

///automatically generated by the FlatBuffers compiler, do not modify
///comm\datalayer
///
///Returns a String as pointer to byte.
METHOD getIdAsBytePtr : POINTER TO BYTE
VAR
	o: UDINT;
END_VAR
o := _offset(vtable_offset:=4);
IF o<>0 THEN
    getIdAsBytePtr := _stringPtr(offset:=o+bb_pos);
ELSE
    getIdAsBytePtr := 0;
END_IF
END_METHOD

///automatically generated by the FlatBuffers compiler, do not modify
///comm\datalayer
///
///Returns a UDINT from the table.
METHOD getProgress : UDINT
VAR
	o: UDINT;
END_VAR
o := _offset(vtable_offset:=8);
IF o<>0 THEN
    getProgress := bb.getUDINT(offset:=o+bb_pos);
ELSE
    getProgress := 0;
END_IF
END_METHOD

///automatically generated by the FlatBuffers compiler, do not modify
///comm\datalayer
///
///Returns a pointer to ProgressData from the table.
METHOD getProgressData : BOOL
VAR_INPUT
	j: UDINT;
	result: POINTER TO comm_datalayer_ProgressData;
END_VAR
VAR
	o: UDINT;
	temp: UDINT;
	temp1: UDINT;
END_VAR
o := _offset(vtable_offset:=14);
IF o<>0 THEN
    temp := _vector(offset:=o);
    temp1 := _indirect(offset:=temp+j*4);
    result^._assign(i:=temp1, _bb:=bb);
    getProgressData := true;
ELSE
    getProgressData := false;
END_IF
END_METHOD

///automatically generated by the FlatBuffers compiler, do not modify
///comm\datalayer
///
///Returns the length of the ProgressData Vector.
METHOD getProgressDataLength : UDINT
VAR
	o: UDINT;
END_VAR
o := _offset(vtable_offset:=14);
IF o<>0 THEN
    getProgressDataLength := _vector_len(offset:=o);
ELSE
    getProgressDataLength := 0;
END_IF
END_METHOD

///automatically generated by the FlatBuffers compiler, do not modify
///comm\datalayer
///
///Returns a String.
METHOD getProgressInfo : STRING
VAR
	o: UDINT;
END_VAR
o := _offset(vtable_offset:=12);
IF o<>0 THEN
    getProgressInfo := _string(offset:=o+bb_pos);
ELSE
    getProgressInfo := '';
END_IF
END_METHOD

///automatically generated by the FlatBuffers compiler, do not modify
///comm\datalayer
///
///Returns a String as pointer to byte.
METHOD getProgressInfoAsBytePtr : POINTER TO BYTE
VAR
	o: UDINT;
END_VAR
o := _offset(vtable_offset:=12);
IF o<>0 THEN
    getProgressInfoAsBytePtr := _stringPtr(offset:=o+bb_pos);
ELSE
    getProgressInfoAsBytePtr := 0;
END_IF
END_METHOD

///automatically generated by the FlatBuffers compiler, do not modify
///comm\datalayer
///
///Returns a pointer to Diagnosis from the table.
METHOD getResult : POINTER TO comm_datalayer_Diagnosis
VAR
	o: UDINT;
	j: UDINT;
END_VAR
o:= _offset(vtable_offset:=10);
IF o<>0 THEN
    j := _indirect(offset:=o+bb_pos);
    result1 := result1._assign(i:=j, _bb:=bb);
    getResult := ADR(result1);
ELSE
    getResult := 0;
END_IF
END_METHOD

///automatically generated by the FlatBuffers compiler, do not modify
///comm\datalayer
///
///Returns a ProgramTask from the ByteBuffer.
/// 
METHOD getRootAsProgramTask : comm_datalayer_ProgramTask
VAR_INPUT
	data: POINTER TO BYTE;
	size: __UXINT;
END_VAR
_bb(data:=data, _capacity:=TO_UDINT(size));
bb REF= _bb;
getRootAsProgramTask := _assign(i:=bb.getUDINT(0), _bb:=bb);
END_METHOD

///automatically generated by the FlatBuffers compiler, do not modify
///comm\datalayer
///
///Returns a BYTE from the table.
METHOD getState : comm_datalayer_ProgramTaskState
VAR
	o: UDINT;
END_VAR
o := _offset(vtable_offset:=6);
IF o<>0 THEN
    getState := bb.getBYTE(offset:=o+bb_pos);
ELSE
    getState := 0;
END_IF
END_METHOD

///automatically generated by the FlatBuffers compiler, do not modify
///comm\datalayer
METHOD keysCompare : DINT
VAR_INPUT
	o1: DINT;
	o2: DINT;
	_bb: REFERENCE TO flatbuffers.ByteBuffer;
END_VAR
keysCompare := compareStrings(_offset_(_bb, 4, o1), _offset_(_bb, 4, o2), _bb);
END_METHOD

///automatically generated by the FlatBuffers compiler, do not modify
///comm\datalayer
///
///Start the table to add values.
METHOD startProgramTask
VAR_INPUT
	builder: REFERENCE TO flatbuffers.FlatBufferBuilder;
END_VAR
_builder REF= builder;
_builder.startTable(numfields:=6);
END_METHOD

///automatically generated by the FlatBuffers compiler, do not modify
///comm\datalayer
///
///Start a vector.
METHOD startProgressDataVector
VAR_INPUT
	builder: REFERENCE TO flatbuffers.FlatBufferBuilder;
	numElems: UDINT;
END_VAR
builder.startVector(elem_size:=4, num_elems:=numElems, alignment:=4);
END_METHOD

///automatically generated by the FlatBuffers compiler, do not modify
///comm\datalayer
METHOD verify : BOOL
VAR_INPUT
	data: POINTER TO BYTE;
	size: __UXINT;
END_VAR
VAR
	_bb: ByteBuffer;
END_VAR
_bb(data:=data, _capacity:=TO_UDINT(size));
verify := verifyProgramTask(data, size, _bb.getUDINT(0));
END_METHOD

///automatically generated by the FlatBuffers compiler, do not modify
///comm\datalayer
{attribute 'conditionalshow' := ''}
METHOD verifyProgramTask : BOOL
VAR_INPUT
	data: POINTER TO BYTE;
	size: __UXINT;
	pointer_: UDINT;
END_VAR
VAR
	_bb: ByteBuffer;
	verifier: flatbuffers.Verifier;
	vt_start: UDINT;
	vt_size: UDINT;
	result1: comm_datalayer_Diagnosis;
	progressData1: comm_datalayer_ProgressData;
	i: DINT;
END_VAR
_bb(data:=data, _capacity:=TO_UDINT(size));
IF pointer_ = 0 THEN
    verifyProgramTask := TRUE;
    RETURN;
END_IF

if pointer_ > (size - SIZEOF(UDINT)) then
    verifyProgramTask := FALSE;
    return;
END_IF

vt_start := _bb.getUDINT(pointer_);
if (pointer_ - vt_start) > (size - SIZEOF(UDINT)) then
    verifyProgramTask := FALSE;
    return;
END_IF

vt_size := _bb.getUINT(pointer_ - vt_start);
verifier(data:=data, size:=size, pointer_:=pointer_, v_size:=vt_size);

IF verifier.verifyTable() AND verifier.verifyString(4) AND verifier.verifyScalar(6) AND verifier.verifyScalar(8) AND result1.verifyDiagnosis(data, size, verifier.getTypeOffset(10)) AND verifier.verifyString(12) AND (verifier.verifyVector_Scalar(14, 4)) THEN
    IF verifier.getTypeOffset(14) <> 0 THEN
        FOR i := 0 TO TO_DINT((_bb.getUDINT(verifier.getTypeOffset(14)) - 1)) DO
            IF NOT progressData1.verifyProgressData(data, size, verifier.getTableVectorOffset(14, TO_UDINT(i))) THEN
                verifyProgramTask := FALSE;
                RETURN;
            END_IF
        END_FOR
    END_IF
    verifyProgramTask := TRUE;
ELSE
    verifyProgramTask := FALSE;
END_IF
END_METHOD

END_FUNCTION_BLOCK

// InternHelpers/comm_datalayer_Diagnosis
///automatically generated by the FlatBuffers compiler, do not modify
///comm\datalayer
///Import FlatBuffers Library
FUNCTION_BLOCK comm_datalayer_Diagnosis EXTENDS flatbuffers.Table
VAR
	_builder: REFERENCE TO flatbuffers.FlatBufferBuilder;
	_bb: flatbuffers.ByteBuffer;
END_VAR

///automatically generated by the FlatBuffers compiler, do not modify
///comm\datalayer
///
///Set the values of a Diagnosis and return it.
{attribute 'conditionalshow' := ''}
METHOD _assign : comm_datalayer_Diagnosis
VAR_INPUT
	i: UDINT;
	_bb: REFERENCE TO flatbuffers.ByteBuffer;
END_VAR
_init(i:=i, _bb:=_bb);
_assign:=this^;
END_METHOD

///automatically generated by the FlatBuffers compiler, do not modify
///comm\datalayer
///
///Set the values of a table.
{attribute 'conditionalshow' := ''}
METHOD _init
VAR_INPUT
	i: UDINT;
	_bb: REFERENCE TO flatbuffers.ByteBuffer;
END_VAR
_reset(i:=i, _bb:=_bb);
END_METHOD

///automatically generated by the FlatBuffers compiler, do not modify
///comm\datalayer
///
///Add values to the table.
METHOD addCause
VAR_INPUT
	causeOffset: UDINT;
END_VAR
IF NOT __ISVALIDREF(_builder) THEN
  SysExceptGenerateException(RTSEXCPT_INVALID_HANDLE);
END_IF
_builder.add_Offset(o:=5, x:=causeOffset, d:=0);
END_METHOD

///automatically generated by the FlatBuffers compiler, do not modify
///comm\datalayer
///
///Add values to the table.
METHOD addDetailedDiagnosisCode
VAR_INPUT
	detailedDiagnosisCode: UDINT;
END_VAR
IF NOT __ISVALIDREF(_builder) THEN
  SysExceptGenerateException(RTSEXCPT_INVALID_HANDLE);
END_IF
_builder.add_UDINT(o:=1, x:=detailedDiagnosisCode, d:=0);
END_METHOD

///automatically generated by the FlatBuffers compiler, do not modify
///comm\datalayer
///
///Add values to the table.
METHOD addDynamicDescription
VAR_INPUT
	dynamicDescriptionOffset: UDINT;
END_VAR
IF NOT __ISVALIDREF(_builder) THEN
  SysExceptGenerateException(RTSEXCPT_INVALID_HANDLE);
END_IF
_builder.add_Offset(o:=2, x:=dynamicDescriptionOffset, d:=0);
END_METHOD

///automatically generated by the FlatBuffers compiler, do not modify
///comm\datalayer
///
///Add values to the table.
METHOD addEntity
VAR_INPUT
	entityOffset: UDINT;
END_VAR
IF NOT __ISVALIDREF(_builder) THEN
  SysExceptGenerateException(RTSEXCPT_INVALID_HANDLE);
END_IF
_builder.add_Offset(o:=3, x:=entityOffset, d:=0);
END_METHOD

///automatically generated by the FlatBuffers compiler, do not modify
///comm\datalayer
///
///Add values to the table.
METHOD addMainDiagnosisCode
VAR_INPUT
	mainDiagnosisCode: UDINT;
END_VAR
IF NOT __ISVALIDREF(_builder) THEN
  SysExceptGenerateException(RTSEXCPT_INVALID_HANDLE);
END_IF
_builder.add_UDINT(o:=0, x:=mainDiagnosisCode, d:=0);
END_METHOD

///automatically generated by the FlatBuffers compiler, do not modify
///comm\datalayer
///
///Add values to the table.
METHOD addMoreInfo
VAR_INPUT
	moreInfoOffset: UDINT;
END_VAR
IF NOT __ISVALIDREF(_builder) THEN
  SysExceptGenerateException(RTSEXCPT_INVALID_HANDLE);
END_IF
_builder.add_Offset(o:=4, x:=moreInfoOffset, d:=0);
END_METHOD

///automatically generated by the FlatBuffers compiler, do not modify
///comm\datalayer
///
///Creates a Vector of the table and returns the offset to it.
METHOD createCauseVector : UDINT
VAR_INPUT
	builder: REFERENCE TO flatbuffers.FlatBufferBuilder;
	data: POINTER TO UDINT;
	size: UDINT;
END_VAR
VAR
	i: DINT;
	temp: POINTER TO UDINT;
END_VAR
IF NOT __ISVALIDREF(builder) THEN
  SysExceptGenerateException(RTSEXCPT_INVALID_HANDLE);
END_IF
builder.startVector(elem_size:=4, num_elems:=size, alignment:=4);
FOR i:=TO_DINT(size-1) TO 0 BY -1 DO
    temp:=data+TO_UDINT(i*4);
    builder.addOffset(off:=temp^);
END_FOR
createCauseVector := builder.endVector();
END_METHOD

///automatically generated by the FlatBuffers compiler, do not modify
///comm\datalayer
///
///Creates a table in the Flatbuffer and returns the offset to it.
METHOD createDiagnosis : UDINT
VAR_INPUT
	builder: REFERENCE TO flatbuffers.FlatBufferBuilder;
	mainDiagnosisCode: UDINT;
	/// Main diagnosis code for diagnosis system. E.g.: 0x3F0A0901
	detailedDiagnosisCode: UDINT;
	/// Detailed diagnosis code for diagnosis system. E.g.: 0xC00E2050
	dynamicDescription: STRING;
	/// A human-readable explanation with even more detailed information specific to this occurrence of the problem.
	entity: STRING;
	/// Resource or entity which causes the problem E.g.: motion/axs/Axis_1
	moreInfoOffset: UDINT;
	/// More information about the diagnosis
	causeOffset: UDINT;
END_VAR
VAR
	dynamicDescriptionOffset: UDINT;
	entityOffset: UDINT;
END_VAR
_builder REF= builder;
IF NOT __ISVALIDREF(_builder) THEN
  SysExceptGenerateException(RTSEXCPT_INVALID_HANDLE);
END_IF
dynamicDescriptionOffset := builder.createString(dynamicDescription);
entityOffset := builder.createString(entity);
_builder.startTable(numfields:=6);
addMainDiagnosisCode(mainDiagnosisCode:=mainDiagnosisCode);
addDetailedDiagnosisCode(detailedDiagnosisCode:=detailedDiagnosisCode);
addDynamicDescription(dynamicDescriptionOffset:=dynamicDescriptionOffset);
addEntity(entityOffset:=entityOffset);
addMoreInfo(moreInfoOffset:=moreInfoOffset);
addCause(causeOffset:=causeOffset);
createDiagnosis := endDiagnosis();
END_METHOD

///automatically generated by the FlatBuffers compiler, do not modify
///comm\datalayer
METHOD createSortedmoreInfoVector : UDINT
VAR_INPUT
	builder: REFERENCE TO flatbuffers.Flatbufferbuilder;
	obj1: REFERENCE TO comm_datalayer_DiagMoreInfo;
	offsets: POINTER TO DINT;
	size: UDINT;
END_VAR
createSortedmoreInfoVector := builder.createSortedVectorOfTables(bb_:=builder.dataBuffer(), obj:=obj1, offsets := offsets, size:=size);
END_METHOD

///automatically generated by the FlatBuffers compiler, do not modify
///comm\datalayer
///
///End the table and return a offset to it
METHOD endDiagnosis : UDINT
VAR
	o: UDINT;
END_VAR
o := _builder.endTable();
_builder REF= 0;
endDiagnosis := o;
END_METHOD

///automatically generated by the FlatBuffers compiler, do not modify
///comm\datalayer
///
///Returns a pointer to Diagnosis from the table.
METHOD getCause : BOOL
VAR_INPUT
	j: UDINT;
	result: POINTER TO comm_datalayer_Diagnosis;
END_VAR
VAR
	o: UDINT;
	temp: UDINT;
	temp1: UDINT;
END_VAR
o := _offset(vtable_offset:=14);
IF o<>0 THEN
    temp := _vector(offset:=o);
    temp1 := _indirect(offset:=temp+j*4);
    result^._assign(i:=temp1, _bb:=bb);
    getCause := true;
ELSE
    getCause := false;
END_IF
END_METHOD

///automatically generated by the FlatBuffers compiler, do not modify
///comm\datalayer
///
///Returns the length of the Cause Vector.
METHOD getCauseLength : UDINT
VAR
	o: UDINT;
END_VAR
o := _offset(vtable_offset:=14);
IF o<>0 THEN
    getCauseLength := _vector_len(offset:=o);
ELSE
    getCauseLength := 0;
END_IF
END_METHOD

///automatically generated by the FlatBuffers compiler, do not modify
///comm\datalayer
///
///Returns a UDINT from the table.
METHOD getDetailedDiagnosisCode : UDINT
VAR
	o: UDINT;
END_VAR
o := _offset(vtable_offset:=6);
IF o<>0 THEN
    getDetailedDiagnosisCode := bb.getUDINT(offset:=o+bb_pos);
ELSE
    getDetailedDiagnosisCode := 0;
END_IF
END_METHOD

///automatically generated by the FlatBuffers compiler, do not modify
///comm\datalayer
///
///Returns a String.
METHOD getDynamicDescription : STRING
VAR
	o: UDINT;
END_VAR
o := _offset(vtable_offset:=8);
IF o<>0 THEN
    getDynamicDescription := _string(offset:=o+bb_pos);
ELSE
    getDynamicDescription := '';
END_IF
END_METHOD

///automatically generated by the FlatBuffers compiler, do not modify
///comm\datalayer
///
///Returns a String as pointer to byte.
METHOD getDynamicDescriptionAsBytePtr : POINTER TO BYTE
VAR
	o: UDINT;
END_VAR
o := _offset(vtable_offset:=8);
IF o<>0 THEN
    getDynamicDescriptionAsBytePtr := _stringPtr(offset:=o+bb_pos);
ELSE
    getDynamicDescriptionAsBytePtr := 0;
END_IF
END_METHOD

///automatically generated by the FlatBuffers compiler, do not modify
///comm\datalayer
///
///Returns a String.
METHOD getEntity : STRING
VAR
	o: UDINT;
END_VAR
o := _offset(vtable_offset:=10);
IF o<>0 THEN
    getEntity := _string(offset:=o+bb_pos);
ELSE
    getEntity := '';
END_IF
END_METHOD

///automatically generated by the FlatBuffers compiler, do not modify
///comm\datalayer
///
///Returns a String as pointer to byte.
METHOD getEntityAsBytePtr : POINTER TO BYTE
VAR
	o: UDINT;
END_VAR
o := _offset(vtable_offset:=10);
IF o<>0 THEN
    getEntityAsBytePtr := _stringPtr(offset:=o+bb_pos);
ELSE
    getEntityAsBytePtr := 0;
END_IF
END_METHOD

///automatically generated by the FlatBuffers compiler, do not modify
///comm\datalayer
///
///Returns a UDINT from the table.
METHOD getMainDiagnosisCode : UDINT
VAR
	o: UDINT;
END_VAR
o := _offset(vtable_offset:=4);
IF o<>0 THEN
    getMainDiagnosisCode := bb.getUDINT(offset:=o+bb_pos);
ELSE
    getMainDiagnosisCode := 0;
END_IF
END_METHOD

///automatically generated by the FlatBuffers compiler, do not modify
///comm\datalayer
///
///Returns a pointer to DiagMoreInfo from the table.
METHOD getMoreInfo : BOOL
VAR_INPUT
	j: UDINT;
	result: POINTER TO comm_datalayer_DiagMoreInfo;
END_VAR
VAR
	o: UDINT;
	temp: UDINT;
	temp1: UDINT;
END_VAR
o := _offset(vtable_offset:=12);
IF o<>0 THEN
    temp := _vector(offset:=o);
    temp1 := _indirect(offset:=temp+j*4);
    result^._assign(i:=temp1, _bb:=bb);
    getMoreInfo := true;
ELSE
    getMoreInfo := false;
END_IF
END_METHOD

///automatically generated by the FlatBuffers compiler, do not modify
///comm\datalayer
///
///Returns the length of the MoreInfo Vector.
METHOD getMoreInfoLength : UDINT
VAR
	o: UDINT;
END_VAR
o := _offset(vtable_offset:=12);
IF o<>0 THEN
    getMoreInfoLength := _vector_len(offset:=o);
ELSE
    getMoreInfoLength := 0;
END_IF
END_METHOD

///automatically generated by the FlatBuffers compiler, do not modify
///comm\datalayer
///
///Returns a Diagnosis from the ByteBuffer.
/// 
METHOD getRootAsDiagnosis : comm_datalayer_Diagnosis
VAR_INPUT
	data: POINTER TO BYTE;
	size: __UXINT;
END_VAR
_bb(data:=data, _capacity:=TO_UDINT(size));
bb REF= _bb;
getRootAsDiagnosis := _assign(i:=bb.getUDINT(0), _bb:=bb);
END_METHOD

///automatically generated by the FlatBuffers compiler, do not modify
///comm\datalayer
///
///Start a vector.
METHOD startCauseVector
VAR_INPUT
	builder: REFERENCE TO flatbuffers.FlatBufferBuilder;
	numElems: UDINT;
END_VAR
builder.startVector(elem_size:=4, num_elems:=numElems, alignment:=4);
END_METHOD

///automatically generated by the FlatBuffers compiler, do not modify
///comm\datalayer
///
///Start the table to add values.
METHOD startDiagnosis
VAR_INPUT
	builder: REFERENCE TO flatbuffers.FlatBufferBuilder;
END_VAR
_builder REF= builder;
_builder.startTable(numfields:=6);
END_METHOD

///automatically generated by the FlatBuffers compiler, do not modify
///comm\datalayer
///
///Start a vector.
METHOD startMoreInfoVector
VAR_INPUT
	builder: REFERENCE TO flatbuffers.FlatBufferBuilder;
	numElems: UDINT;
END_VAR
builder.startVector(elem_size:=4, num_elems:=numElems, alignment:=4);
END_METHOD

///automatically generated by the FlatBuffers compiler, do not modify
///comm\datalayer
METHOD verify : BOOL
VAR_INPUT
	data: POINTER TO BYTE;
	size: __UXINT;
END_VAR
VAR
	_bb: ByteBuffer;
END_VAR
_bb(data:=data, _capacity:=TO_UDINT(size));
verify := verifyDiagnosis(data, size, _bb.getUDINT(0));
END_METHOD

///automatically generated by the FlatBuffers compiler, do not modify
///comm\datalayer
{attribute 'conditionalshow' := ''}
METHOD verifyDiagnosis : BOOL
VAR_INPUT
	data: POINTER TO BYTE;
	size: __UXINT;
	pointer_: UDINT;
END_VAR
VAR
	_bb: ByteBuffer;
	verifier: flatbuffers.Verifier;
	vt_start: UDINT;
	vt_size: UDINT;
	moreInfo1: comm_datalayer_DiagMoreInfo;
	i: DINT;
	cause1: comm_datalayer_Diagnosis;
END_VAR
_bb(data:=data, _capacity:=TO_UDINT(size));
IF pointer_ = 0 THEN
    verifyDiagnosis := TRUE;
    RETURN;
END_IF

if pointer_ > (size - SIZEOF(UDINT)) then
    verifyDiagnosis := FALSE;
    return;
END_IF

vt_start := _bb.getUDINT(pointer_);
if (pointer_ - vt_start) > (size - SIZEOF(UDINT)) then
    verifyDiagnosis := FALSE;
    return;
END_IF

vt_size := _bb.getUINT(pointer_ - vt_start);
verifier(data:=data, size:=size, pointer_:=pointer_, v_size:=vt_size);

IF verifier.verifyTable() AND verifier.verifyScalar(4) AND verifier.verifyScalar(6) AND verifier.verifyString(8) AND verifier.verifyString(10) AND (verifier.verifyVector_Scalar(12, 4)) AND (verifier.verifyVector_Scalar(14, 4)) THEN
    IF verifier.getTypeOffset(12) <> 0 THEN
        FOR i := 0 TO TO_DINT((_bb.getUDINT(verifier.getTypeOffset(12)) - 1)) DO
            IF NOT moreInfo1.verifyDiagMoreInfo(data, size, verifier.getTableVectorOffset(12, TO_UDINT(i))) THEN
                verifyDiagnosis := FALSE;
                RETURN;
            END_IF
        END_FOR
    END_IF
    IF verifier.getTypeOffset(14) <> 0 THEN
        FOR i := 0 TO TO_DINT((_bb.getUDINT(verifier.getTypeOffset(14)) - 1)) DO
            IF NOT cause1.verifyDiagnosis(data, size, verifier.getTableVectorOffset(14, TO_UDINT(i))) THEN
                verifyDiagnosis := FALSE;
                RETURN;
            END_IF
        END_FOR
    END_IF
    verifyDiagnosis := TRUE;
ELSE
    verifyDiagnosis := FALSE;
END_IF
END_METHOD

END_FUNCTION_BLOCK

// InternHelpers/comm_datalayer_DiagMoreInfo
///automatically generated by the FlatBuffers compiler, do not modify
///comm\datalayer
///Import FlatBuffers Library
FUNCTION_BLOCK comm_datalayer_DiagMoreInfo EXTENDS flatbuffers.Table
VAR
	_builder: REFERENCE TO flatbuffers.FlatBufferBuilder;
	_bb: flatbuffers.ByteBuffer;
END_VAR

///automatically generated by the FlatBuffers compiler, do not modify
///comm\datalayer
///
///Set the values of a DiagMoreInfo and return it.
{attribute 'conditionalshow' := ''}
METHOD _assign : comm_datalayer_DiagMoreInfo
VAR_INPUT
	i: UDINT;
	_bb: REFERENCE TO flatbuffers.ByteBuffer;
END_VAR
_init(i:=i, _bb:=_bb);
_assign:=this^;
END_METHOD

///automatically generated by the FlatBuffers compiler, do not modify
///comm\datalayer
///
///Set the values of a table.
{attribute 'conditionalshow' := ''}
METHOD _init
VAR_INPUT
	i: UDINT;
	_bb: REFERENCE TO flatbuffers.ByteBuffer;
END_VAR
_reset(i:=i, _bb:=_bb);
END_METHOD

///automatically generated by the FlatBuffers compiler, do not modify
///comm\datalayer
///
///Add values to the table.
METHOD addKey
VAR_INPUT
	keyOffset: UDINT;
END_VAR
IF NOT __ISVALIDREF(_builder) THEN
  SysExceptGenerateException(RTSEXCPT_INVALID_HANDLE);
END_IF
_builder.add_Offset(o:=0, x:=keyOffset, d:=0);
END_METHOD

///automatically generated by the FlatBuffers compiler, do not modify
///comm\datalayer
///
///Add values to the table.
METHOD addValue
VAR_INPUT
	valueOffset: UDINT;
END_VAR
IF NOT __ISVALIDREF(_builder) THEN
  SysExceptGenerateException(RTSEXCPT_INVALID_HANDLE);
END_IF
_builder.add_Offset(o:=1, x:=valueOffset, d:=0);
END_METHOD

///automatically generated by the FlatBuffers compiler, do not modify
///comm\datalayer
///
///Creates a table in the Flatbuffer and returns the offset to it.
METHOD createDiagMoreInfo : UDINT
VAR_INPUT
	builder: REFERENCE TO flatbuffers.FlatBufferBuilder;
	key: STRING;
	/// defined key 
	///   "requiredLicenses": list of required licences seperated by ","
	///   "requiredScopes": list of required scopes seperated by ","
	value: STRING;
END_VAR
VAR
	keyOffset: UDINT;
	valueOffset: UDINT;
END_VAR
_builder REF= builder;
IF NOT __ISVALIDREF(_builder) THEN
  SysExceptGenerateException(RTSEXCPT_INVALID_HANDLE);
END_IF
keyOffset := builder.createString(key);
valueOffset := builder.createString(value);
_builder.startTable(numfields:=2);
addKey(keyOffset:=keyOffset);
addValue(valueOffset:=valueOffset);
createDiagMoreInfo := endDiagMoreInfo();
END_METHOD

///automatically generated by the FlatBuffers compiler, do not modify
///comm\datalayer
///
///End the table and return a offset to it
METHOD endDiagMoreInfo : UDINT
VAR
	o: UDINT;
END_VAR
o := _builder.endTable();
_builder REF= 0;
endDiagMoreInfo := o;
END_METHOD

///automatically generated by the FlatBuffers compiler, do not modify
///comm\datalayer
///
///Returns a String.
METHOD getKey : STRING
VAR
	o: UDINT;
END_VAR
o := _offset(vtable_offset:=4);
IF o<>0 THEN
    getKey := _string(offset:=o+bb_pos);
ELSE
    getKey := '';
END_IF
END_METHOD

///automatically generated by the FlatBuffers compiler, do not modify
///comm\datalayer
///
///Returns a String as pointer to byte.
METHOD getKeyAsBytePtr : POINTER TO BYTE
VAR
	o: UDINT;
END_VAR
o := _offset(vtable_offset:=4);
IF o<>0 THEN
    getKeyAsBytePtr := _stringPtr(offset:=o+bb_pos);
ELSE
    getKeyAsBytePtr := 0;
END_IF
END_METHOD

///automatically generated by the FlatBuffers compiler, do not modify
///comm\datalayer
///
///Returns a DiagMoreInfo from the ByteBuffer.
/// 
METHOD getRootAsDiagMoreInfo : comm_datalayer_DiagMoreInfo
VAR_INPUT
	data: POINTER TO BYTE;
	size: __UXINT;
END_VAR
_bb(data:=data, _capacity:=TO_UDINT(size));
bb REF= _bb;
getRootAsDiagMoreInfo := _assign(i:=bb.getUDINT(0), _bb:=bb);
END_METHOD

///automatically generated by the FlatBuffers compiler, do not modify
///comm\datalayer
///
///Returns a String.
METHOD getValue : STRING
VAR
	o: UDINT;
END_VAR
o := _offset(vtable_offset:=6);
IF o<>0 THEN
    getValue := _string(offset:=o+bb_pos);
ELSE
    getValue := '';
END_IF
END_METHOD

///automatically generated by the FlatBuffers compiler, do not modify
///comm\datalayer
///
///Returns a String as pointer to byte.
METHOD getValueAsBytePtr : POINTER TO BYTE
VAR
	o: UDINT;
END_VAR
o := _offset(vtable_offset:=6);
IF o<>0 THEN
    getValueAsBytePtr := _stringPtr(offset:=o+bb_pos);
ELSE
    getValueAsBytePtr := 0;
END_IF
END_METHOD

///automatically generated by the FlatBuffers compiler, do not modify
///comm\datalayer
METHOD keysCompare : DINT
VAR_INPUT
	o1: DINT;
	o2: DINT;
	_bb: REFERENCE TO flatbuffers.ByteBuffer;
END_VAR
keysCompare := compareStrings(_offset_(_bb, 4, o1), _offset_(_bb, 4, o2), _bb);
END_METHOD

///automatically generated by the FlatBuffers compiler, do not modify
///comm\datalayer
///
///Start the table to add values.
METHOD startDiagMoreInfo
VAR_INPUT
	builder: REFERENCE TO flatbuffers.FlatBufferBuilder;
END_VAR
_builder REF= builder;
_builder.startTable(numfields:=2);
END_METHOD

///automatically generated by the FlatBuffers compiler, do not modify
///comm\datalayer
{attribute 'conditionalshow' := ''}
METHOD verify : BOOL
VAR_INPUT
	data: POINTER TO BYTE;
	size: __UXINT;
END_VAR
VAR
	_bb: ByteBuffer;
END_VAR
_bb(data:=data, _capacity:=TO_UDINT(size));
verify := verifyDiagMoreInfo(data, size, _bb.getUDINT(0));
END_METHOD

///automatically generated by the FlatBuffers compiler, do not modify
///comm\datalayer
{attribute 'conditionalshow' := ''}
METHOD verifyDiagMoreInfo : BOOL
VAR_INPUT
	data: POINTER TO BYTE;
	size: __UXINT;
	pointer_: UDINT;
END_VAR
VAR
	_bb: ByteBuffer;
	verifier: flatbuffers.Verifier;
	vt_start: UDINT;
	vt_size: UDINT;
END_VAR
_bb(data:=data, _capacity:=TO_UDINT(size));
IF pointer_ = 0 THEN
    verifyDiagMoreInfo := TRUE;
    RETURN;
END_IF

if pointer_ > (size - SIZEOF(UDINT)) then
    verifyDiagMoreInfo := FALSE;
    return;
END_IF

vt_start := _bb.getUDINT(pointer_);
if (pointer_ - vt_start) > (size - SIZEOF(UDINT)) then
    verifyDiagMoreInfo := FALSE;
    return;
END_IF

vt_size := _bb.getUINT(pointer_ - vt_start);
verifier(data:=data, size:=size, pointer_:=pointer_, v_size:=vt_size);

IF verifier.verifyTable() AND verifier.verifyString(4) AND verifier.verifyString(6) THEN
    verifyDiagMoreInfo := TRUE;
ELSE
    verifyDiagMoreInfo := FALSE;
END_IF
END_METHOD

END_FUNCTION_BLOCK

// InternHelpers/comm_datalayer_ProgressData
///automatically generated by the FlatBuffers compiler, do not modify
///comm\datalayer
///Import FlatBuffers Library
FUNCTION_BLOCK comm_datalayer_ProgressData EXTENDS flatbuffers.Table
VAR
	_builder: REFERENCE TO flatbuffers.FlatBufferBuilder;
	_bb: flatbuffers.ByteBuffer;
END_VAR

///automatically generated by the FlatBuffers compiler, do not modify
///comm\datalayer
///
///Set the values of a ProgressData and return it.
{attribute 'conditionalshow' := ''}
METHOD _assign : comm_datalayer_ProgressData
VAR_INPUT
	i: UDINT;
	_bb: REFERENCE TO flatbuffers.ByteBuffer;
END_VAR
_init(i:=i, _bb:=_bb);
_assign:=this^;
END_METHOD

///automatically generated by the FlatBuffers compiler, do not modify
///comm\datalayer
///
///Set the values of a table.
{attribute 'conditionalshow' := ''}
METHOD _init
VAR_INPUT
	i: UDINT;
	_bb: REFERENCE TO flatbuffers.ByteBuffer;
END_VAR
_reset(i:=i, _bb:=_bb);
END_METHOD

///automatically generated by the FlatBuffers compiler, do not modify
///comm\datalayer
///
///Add values to the table.
METHOD addKey
VAR_INPUT
	keyOffset: UDINT;
END_VAR
IF NOT __ISVALIDREF(_builder) THEN
  SysExceptGenerateException(RTSEXCPT_INVALID_HANDLE);
END_IF
_builder.add_Offset(o:=0, x:=keyOffset, d:=0);
END_METHOD

///automatically generated by the FlatBuffers compiler, do not modify
///comm\datalayer
///
///Add values to the table.
METHOD addValue
VAR_INPUT
	valueOffset: UDINT;
END_VAR
IF NOT __ISVALIDREF(_builder) THEN
  SysExceptGenerateException(RTSEXCPT_INVALID_HANDLE);
END_IF
_builder.add_Offset(o:=1, x:=valueOffset, d:=0);
END_METHOD

///automatically generated by the FlatBuffers compiler, do not modify
///comm\datalayer
///
///Creates a table in the Flatbuffer and returns the offset to it.
METHOD createProgressData : UDINT
VAR_INPUT
	builder: REFERENCE TO flatbuffers.FlatBufferBuilder;
	key: STRING;
	value: STRING;
END_VAR
VAR
	keyOffset: UDINT;
	valueOffset: UDINT;
END_VAR
_builder REF= builder;
IF NOT __ISVALIDREF(_builder) THEN
  SysExceptGenerateException(RTSEXCPT_INVALID_HANDLE);
END_IF
keyOffset := builder.createString(key);
valueOffset := builder.createString(value);
_builder.startTable(numfields:=2);
addKey(keyOffset:=keyOffset);
addValue(valueOffset:=valueOffset);
createProgressData := endProgressData();
END_METHOD

///automatically generated by the FlatBuffers compiler, do not modify
///comm\datalayer
///
///End the table and return a offset to it
METHOD endProgressData : UDINT
VAR
	o: UDINT;
END_VAR
o := _builder.endTable();
_builder REF= 0;
endProgressData := o;
END_METHOD

///automatically generated by the FlatBuffers compiler, do not modify
///comm\datalayer
///
///Returns a String.
METHOD getKey : STRING
VAR
	o: UDINT;
END_VAR
o := _offset(vtable_offset:=4);
IF o<>0 THEN
    getKey := _string(offset:=o+bb_pos);
ELSE
    getKey := '';
END_IF
END_METHOD

///automatically generated by the FlatBuffers compiler, do not modify
///comm\datalayer
///
///Returns a String as pointer to byte.
METHOD getKeyAsBytePtr : POINTER TO BYTE
VAR
	o: UDINT;
END_VAR
o := _offset(vtable_offset:=4);
IF o<>0 THEN
    getKeyAsBytePtr := _stringPtr(offset:=o+bb_pos);
ELSE
    getKeyAsBytePtr := 0;
END_IF
END_METHOD

///automatically generated by the FlatBuffers compiler, do not modify
///comm\datalayer
///
///Returns a ProgressData from the ByteBuffer.
/// 
METHOD getRootAsProgressData : comm_datalayer_ProgressData
VAR_INPUT
	data: POINTER TO BYTE;
	size: __UXINT;
END_VAR
_bb(data:=data, _capacity:=TO_UDINT(size));
bb REF= _bb;
getRootAsProgressData := _assign(i:=bb.getUDINT(0), _bb:=bb);
END_METHOD

///automatically generated by the FlatBuffers compiler, do not modify
///comm\datalayer
///
///Returns a String.
METHOD getValue : STRING
VAR
	o: UDINT;
END_VAR
o := _offset(vtable_offset:=6);
IF o<>0 THEN
    getValue := _string(offset:=o+bb_pos);
ELSE
    getValue := '';
END_IF
END_METHOD

///automatically generated by the FlatBuffers compiler, do not modify
///comm\datalayer
///
///Returns a String as pointer to byte.
METHOD getValueAsBytePtr : POINTER TO BYTE
VAR
	o: UDINT;
END_VAR
o := _offset(vtable_offset:=6);
IF o<>0 THEN
    getValueAsBytePtr := _stringPtr(offset:=o+bb_pos);
ELSE
    getValueAsBytePtr := 0;
END_IF
END_METHOD

///automatically generated by the FlatBuffers compiler, do not modify
///comm\datalayer
METHOD keysCompare : DINT
VAR_INPUT
	o1: DINT;
	o2: DINT;
	_bb: REFERENCE TO flatbuffers.ByteBuffer;
END_VAR
keysCompare := compareStrings(_offset_(_bb, 4, o1), _offset_(_bb, 4, o2), _bb);
END_METHOD

///automatically generated by the FlatBuffers compiler, do not modify
///comm\datalayer
///
///Start the table to add values.
METHOD startProgressData
VAR_INPUT
	builder: REFERENCE TO flatbuffers.FlatBufferBuilder;
END_VAR
_builder REF= builder;
_builder.startTable(numfields:=2);
END_METHOD

///automatically generated by the FlatBuffers compiler, do not modify
///comm\datalayer
{attribute 'conditionalshow' := ''}
METHOD verify : BOOL
VAR_INPUT
	data: POINTER TO BYTE;
	size: __UXINT;
END_VAR
VAR
	_bb: ByteBuffer;
END_VAR
_bb(data:=data, _capacity:=TO_UDINT(size));
verify := verifyProgressData(data, size, _bb.getUDINT(0));
END_METHOD

